METHOD checkChildAlmClass : BOOL
//------------------------------------------------------------------------------------------------------
// check child alarm classes
// set me alarm class active if at least one child has an EOFF
IF CheckAllChildAlmClass(E_AlmClass.EOFF) THEN
	CIf.Job.eMe_ActivAlmClass := E_AlmClass.EOFF;
	me.Alarm.bolfp := TRUE;
ELSIF CheckAllChildAlmClass(E_AlmClass.OFF) THEN
	CIf.Job.eMe_ActivAlmClass := E_AlmClass.OFF;
	me.Alarm.bolfp := TRUE;
ELSIF CheckAllChildAlmClass(E_AlmClass.STOP) THEN  // FB_MER needs alarm class STOP
	CIf.Job.eMe_ActivAlmClass := E_AlmClass.STOP;
	me.Alarm.bolfp := TRUE;
ELSE
	IF (me.Alarm.bolfp) THEN
		CIf.Job.eMe_ActivAlmClass := E_AlmClass.NONE; // no reset necessary
		me.Alarm.bolfp := FALSE;
	END_IF
END_IF

//------------------------------------------------------------------------------------------------------
// set alarm class parent of childs
//------------------------------------------------------------------------------------------------------
// set alarm class parent of childs in the case of a parent EOFF or me=OFF or EOFF
IF (CIf.Job.eParent_ActivAlmClass=E_AlmClass.EOFF) THEN
	SetAllChildAlmClass(CIf.Job.eParent_ActivAlmClass);
ELSIF(CIf.Job.eMe_ActivAlmClass=E_AlmClass.EOFF) OR (CIf.Job.eMe_ActivAlmClass=E_AlmClass.OFF) THEN
	SetAllChildAlmClass(CIf.Job.eMe_ActivAlmClass);
ELSE
	// no important alarm for child active
	SetAllChildAlmClass(E_AlmClass.NONE);
END_IF
END_METHOD

METHOD PROTECTED checkChildValid : BOOL
IF (usiNumOfLines = usiNumOfValidPointerToLine) THEN
	checkChildValid:= TRUE;
ELSE
	checkChildValid:= FALSE;
	// Invalid child pointer
	IF (usiNumOfLines <> usiNumOfValidPointerToLine) THEN
		// SIf.Alm[1].strText := 'Invalid child pointer'; 
		pfbAlarmCtrl^.setAlarm(CIf.Info.intCtrlId,1,0,ADR(SIf.Alm),E_AlmState.RST,CIf.Job.eMe_ActivAlmClass);	
	END_IF
END_IF
END_METHOD

METHOD PROTECTED checkStateAllLines : BOOL
VAR_INPUT
	cSTA: INT;
END_VAR
VAR
	ii: INT;
	usiNumOfCheckedChilds: USINT;
END_VAR
// Method check input state of all lines

//Init
checkStateAllLines:= FALSE;
usiNumOfCheckedChilds:= 0;

// Loop over all childs
FOR ii:=0 TO usiNumOfLines-1 BY 1 DO
	// Check state	
	// Special condition: In case if the child is in state ERROR and STOP is requested. Set child as checked.
	// Parent controller need state STOP that automatic stop sequence can work for all other childs.
	IF (a_pLineChildCIF[ii]^.Job.intState = cSTA) OR ((a_pLineChildCIF[ii]^.Job.intState = cSTA_ERROR) AND (cSTA = cSTA_STOP)) THEN
		usiNumOfCheckedChilds:= usiNumOfCheckedChilds+1;
		SIf.Cur.a_bolChildReady[ii] := TRUE;
	ELSE
		SIf.Cur.a_bolChildReady[ii] := FALSE;		
	END_IF

END_FOR

// All states equal the input state
IF (usiNumOfCheckedChilds = usiNumOfLines) THEN
	checkStateAllLines:= TRUE;
END_IF
END_METHOD

METHOD PROTECTED CmdToAllLines
VAR_INPUT
	cCMD: INT;
END_VAR
VAR
	ii: INT;
END_VAR
// Method send input command to all existing line child controller.
FOR ii:=0 TO usiNumOfLines-1 BY 1 DO	
	a_pLineChildCIF[ii]^.Job.intACmd:= cCMD;
END_FOR
END_METHOD

METHOD PROTECTED CtrlInit : BOOL
VAR
	ii: INT;
END_VAR
SUPER^.CtrlInit();

//----------------------------------------------------------------------
// Initialize all lines
//----------------------------------------------------------------------

// Method initialize all line child controller.
FOR ii:=0 TO usiNumOfLines-1 BY 1 DO	
	a_pLineChildCIF[ii] := THIS^.AddChild(a_pLineChildCtrl[ii]^);
	a_pLineChildSIF[ii] := a_pLineChildCtrl[ii]^.getCtrlSIf();
END_FOR
END_METHOD

METHOD FB_init : BOOL
VAR_INPUT
	///if TRUE, the retain variables are initialized (warm start / cold start)
	bInitRetains: BOOL;
	///if TRUE, the instance afterwards gets moved into the copy code (online change)
	bInCopyCode: BOOL;
END_VAR
VAR
	ii: UINT;
END_VAR
//------------------------------------------------------------------------------------------------------------------------
// to manually change in new FUB implementation!!!
// define valid commands for this controller
FOR ii:= 0 TO (SIZEOF(CIf.Job.aCmdList)/SIZEOF(CIf.Job.aCmdList[0])-1) BY 1 DO
	IF (CIf.Job.aCmdList[ii].intCmd=cCMD_INITIALIZED) THEN
		// found first empty array element
		EXIT;
	END_IF
END_FOR

CIf.Job.aCmdList[ii].intCmd := cCMD_STOP;
CIf.Job.aCmdList[ii].strName := 'Stop'; 
CIf.Job.aCmdList[ii].bolAvailable := TRUE;
ii := ii +1;
CIf.Job.aCmdList[ii].intCmd := cCMD_RUN;
CIf.Job.aCmdList[ii].strName := 'Run';
CIf.Job.aCmdList[ii].bolAvailable := TRUE;

// set name of class/typ
CIf.Info.strType := 'FB_MER'; 

// set alarm class
SIf.Alm[1].eAlmClass := E_AlmClass.STOP;
SIf.Alm[1].strText := 'Invalid child pointer';
SIf.Alm[2].eAlmClass := E_AlmClass.INFO;
SIf.Alm[2].strText := 'Invalid line number. Line not exist';
SIf.Alm[3].eAlmClass := E_AlmClass.INFO;
SIf.Alm[3].strText := 'Merger waits for jam sensor free'; 


//*******************************************************************************
// initial values
//*******************************************************************************

// software configuration
CIf.SwCfg.bolExist := TRUE;
CIf.SwCfg.bolSimulation := FALSE;

// configuration
SIf.Cfg.usiMergeMainMode:= E_Typ_MER_MODE.Automatic;
SIf.Cfg.usiCountJamSensors:= 0;

// parameter
SIf.Par.udi_jamTimeout_ms:= 500;
FOR ii:= 0 TO Base_PLC.cMaxNrOfChilds DO
	SIf.Par.a_bolEnableHangerRelease[ii] := TRUE;
END_FOR
// Default parameter for the lines are set in method InitLines
END_METHOD

METHOD PROTECTED getCmdState : STRING
VAR_INPUT
	intCmdState: INT;
	bolState: BOOL;
END_VAR
getCmdState := SUPER^.getCmdState(intCmdState:=intCmdState,bolState:=bolState); // get global/base defined cmds/states
IF (getCmdState='') THEN // global not defined get local
	// get string cmd/state string information in runtime
	IF (bolState=FALSE) THEN
		// cmd's
		CASE intCmdState OF
		END_CASE;
	ELSE
	
	// states
		CASE intCmdState OF	
			// SUB States
			cSTA_SUB_INITIALIZED:
				getCmdState := 'cSTA_SUB_INITIALIZED';			
			cSTA_SUB_WAIT_FOR_CMD:
				getCmdState := 'cSTA_SUB_WAIT_FOR_CMD';					
			cSTA_SUB_CHECK_HANGER_EXIST:
				getCmdState := 'cSTA_SUB_CHECK_HANGER_EXIST';
			cSTA_SUB_SEND_RELEASE:
				getCmdState := 'cSTA_SUB_SEND_RELEASE';
			cSTA_SUB_SEND_RELEASE_ALL:
				getCmdState := 'cSTA_SUB_SEND_RELEASE_ALL';	
			cSTA_SUB_SEND_STOP:
				getCmdState := 'cSTA_SUB_SEND_STOP';		
			cSTA_SUB_WAIT_JOB_DONE:
				getCmdState := 'cSTA_SUB_WAIT_JOB_DONE';
			cSTA_SUB_CHECK_MERGE_CON:
				getCmdState := 'cSTA_SUB_CHECK_MERGE_CON';
			cSTA_SUB_WAIT_LINE_FREE:
				getCmdState := 'cSTA_SUB_WAIT_LINE_FREE';	
			cSTA_SUB_END:
				getCmdState := 'cSTA_SUB_END';	
		END_CASE;
	END_IF
END_IF
END_METHOD

METHOD getCtrlSIf : POINTER TO T_Ctrl_SIf_MER
getCtrlSIf := ADR(SIf);
END_METHOD

METHOD PROTECTED IoInBridge : BOOL
// digitale and analoge inputs read from hardware or forcing
// Read sensors for waiting if a jam is detected
FOR intI := 1 TO SIf.Cfg.usiCountJamSensors DO
	SIf.In.a_bolJamSensor[intI].map := THIS^.In_a_bolJamSensor[intI];
	IF (CIf.SwCfg.bolSimulation = FALSE) THEN
		getInBol(CIf.Job.bolIoForce,ADR(SIf.In.a_bolJamSensor[intI]));
	END_IF
END_FOR

IF (CIf.SwCfg.bolSimulation = FALSE) THEN
	//ctrl.In.bol_PosSwitchBasicDefTyp.intern := getInBol(ctrl.ifc.Job.bol_Force ,ADR(ctrl.In.bol_PosSwitchBasicDefTyp);
ELSE
	//simulation of global IO
END_IF
END_METHOD

METHOD PROTECTED IoOutBridge : BOOL
// digitale and analoge inputs read from hardware or forcing

// ... no physical outputs

IF (CIf.SwCfg.bolSimulation = FALSE) THEN
	// check interlocks to prevent damages
	IF (CIf.Job.bolIlkOverwrite=FALSE) THEN
		;
	END_IF
END_IF
END_METHOD

PROPERTY MaxCapacity : DINT
GET
MaxCapacity:= SIf.Cur.dinMaxCapacity;
END_GET
END_PROPERTY

PROPERTY NumOfHangers : DINT
GET
NumOfHangers:= SIf.Cur.dinCurrentItemCount;
END_GET
END_PROPERTY

METHOD PROTECTED sta_OFF : BOOL
// state implemetation
//--------------------------------------------------------------------------------------
// Entry action
	IF (me.StateMachine.intState<>me.StateMachine.intStateLastCycle) THEN
		me.StateMachine.intStateLastCycle := me.StateMachine.intState;
		;		
	END_IF

//--------------------------------------------------------------------------------------
// Cyclic action
	IF (me.StateMachine.intState=me.StateMachine.intStateLastCycle) THEN
		
		// Reset total counter
		SIf.Cur.dinNumOfMergedHangersTotal:= 0;
		
		// State Change Condition
		IF (me.Alarm.eActivAlmClass<>E_AlmClass.EOFF) AND (me.Alarm.eActivAlmClass<>E_AlmClass.OFF) THEN
			IF (me.intCmd=cCMD_STOP) THEN
				me.StateMachine.intStateNext := cSTA_STOPBusy;
			ELSIF (me.intCmd=cCMD_RUN) THEN 
				me.StateMachine.intStateNext := cSTA_RUNBusy;
			END_IF
		END_IF
	END_IF

//--------------------------------------------------------------------------------------
// Exit action
	IF (me.StateMachine.intState<>me.StateMachine.intStateNext) THEN
		;
	END_IF
END_METHOD

METHOD PROTECTED sta_RUN : BOOL
// state implemetation
//--------------------------------------------------------------------------------------
// Entry action
	IF (me.StateMachine.intState<>me.StateMachine.intStateLastCycle) THEN
		me.StateMachine.intStateLastCycle := me.StateMachine.intState;	
		;
	END_IF

//--------------------------------------------------------------------------------------
// Cyclic action
	IF (me.StateMachine.intState=me.StateMachine.intStateLastCycle) THEN
			
	
		// Check States for parent information
		THIS^.checkStateAllLines(cSTA_RUN);

		// Check jam detection
		IF (udiJamReleaseDelayTime_ms > SIf.Par.udi_jamTimeout_ms) THEN
			bolJamDetected := FALSE;
		ELSE
			udiJamReleaseDelayTime_ms := udiJamReleaseDelayTime_ms + me.FUBInfo.udiSample_ms;
		END_IF
		
		FOR intI := 1 TO SIf.Cfg.usiCountJamSensors DO
			// Start jam timer
			IF ((SIf.In.a_bolJamSensor[intI].intern = TRUE) AND (a_bolJamSensorOnce[intI] = FALSE)) THEN
				a_bolJamSensorOnce[intI]:= TRUE;
				//a_udiTimeJamDetection[intI]:= me.StateMachine.udiTimeInState_ms;
				a_udiTimeJamDetection[intI]:= 0;
			// Stop jam timer
			ELSIF ((SIf.In.a_bolJamSensor[intI].intern = FALSE) AND (a_bolJamSensorOnce[intI] = TRUE)) THEN
				a_bolJamSensorOnce[intI]:= FALSE;
			// Set flag if neccessary
			ELSIF ((SIf.In.a_bolJamSensor[intI].intern = TRUE) AND (a_bolJamSensorOnce[intI] = TRUE)) THEN
				//IF (me.StateMachine.udiTimeInState_ms > a_udiTimeJamDetection[intI] + SIf.Par.udi_jamTimeout_ms) THEN
				IF (a_udiTimeJamDetection[intI] > SIf.Par.udi_jamTimeout_ms) THEN
					bolJamDetected := TRUE;
					udiJamReleaseDelayTime_ms := 0;
				END_IF
			END_IF
			a_udiTimeJamDetection[intI]:= a_udiTimeJamDetection[intI]+ me.FUBInfo.udiSample_ms;
		END_FOR
	
		//----------------------------------------------------------------------------------------
		// Substates for merging lines dependent time or distribution of the number of hangers
		//----------------------------------------------------------------------------------------
		CASE me.SubStateMachine.intState OF
	
			//-----------------------------------------------
			// INITIALIZE 					(MODE: All modes)
			//-----------------------------------------------
			cSTA_SUB_INITIALIZED:
			
				// Check configured main mode
				CASE SIf.Cfg.usiMergeMainMode OF	
				
					// Mode - Automatic
					E_Typ_MER_MODE.Automatic:		
						me.SubStateMachine.intStateNext := cSTA_SUB_CHECK_HANGER_EXIST;					
									
					// Mode - OnCommand	
					E_Typ_MER_MODE.OnCommand:		
						me.SubStateMachine.intStateNext := cSTA_SUB_WAIT_FOR_CMD;
														
				END_CASE
			
			//-----------------------------------------------
			// WAIT FOR COMMAND 			(MODE: OnCommand)
			//-----------------------------------------------	
			cSTA_SUB_WAIT_FOR_CMD:
			
				// Wait for command to release all
				IF (me.intCmd=SLB_CmdState.cCMD_RELEASE_ALL) THEN
					// Check about valid line number
					IF ((SIf.Par.usiLineNumToReleaseAll = 0) OR (SIf.Par.usiLineNumToReleaseAll > usiNumOfLines)) THEN
						// Invalid line	
						// SIf.Alm[2].strText := 'Invalid line number. Line not exist'; 
						pfbAlarmCtrl^.setAlarm(CIf.Info.intCtrlId,2,0,ADR(SIf.Alm),E_AlmState.RST,CIf.Job.eMe_ActivAlmClass);		
					ELSE
						// Valid line	
						usiLineNumToReleaseAll:= SIf.Par.usiLineNumToReleaseAll-1;
						me.SubStateMachine.intStateNext := cSTA_SUB_SEND_RELEASE_ALL;
					END_IF
						
				END_IF
				
			//-----------------------------------------------
			// CHECK HANGER EXIST 			(MODE: Automatic)     
			//-----------------------------------------------
			cSTA_SUB_CHECK_HANGER_EXIST:
				// Entry action
				IF (me.SubStateMachine.intState<>me.SubStateMachine.intStateLastCycle) THEN
					me.SubStateMachine.intStateLastCycle := me.SubStateMachine.intState;							
					;						
				END_IF
				
				// Init
				bolReleaseHanger:= FALSE;
					
				// Check hanger exists on line
				IF (a_pLineChildSIF[usiIndexToRelease]^.Cur.bolHangerDetected=TRUE) AND 
					(Sif.par.a_bolEnableHangerRelease[usiIndexToRelease] = TRUE) THEN		// MRU added
					bolReleaseHanger:= TRUE;					
				ELSE		
					// No hanger on this line, check next
					IF (usiIndexToRelease < (usiNumOfLines-1)) THEN
						// Inc. index to next line
						usiIndexToRelease:= usiIndexToRelease + 1;	
					ELSE
						usiIndexToRelease:= 0;
					END_IF
				END_IF			
	
				// State Change Condition
				IF (bolReleaseHanger=TRUE) THEN
					me.SubStateMachine.intStateNext := cSTA_SUB_SEND_RELEASE;
					// Reset counter and timer
					dinNumOfPassedHangers:=0;
					udiMergingTime:=0;
				END_IF
					
			//-----------------------------------------------
			// SEND RELEASE					(MODE: Automatic)
			//-----------------------------------------------
			cSTA_SUB_SEND_RELEASE:		
	
				// Send release command to line X (trigger command)
				a_pLineChildCIF[usiIndexToRelease]^.Job.intACmd:= STB_CmdState.cCMD_RELEASE;				
				
				// State Change Condition
				IF(TRUE)THEN
					me.SubStateMachine.intStateNext := cSTA_SUB_WAIT_JOB_DONE;					
				END_IF	
						
			//-----------------------------------------------
			// SEND RELEASE	ALL				(MODE: OnCommand)
			//-----------------------------------------------
			cSTA_SUB_SEND_RELEASE_ALL:
			
				// Send release all command to line X
				a_pLineChildCIF[usiLineNumToReleaseAll]^.Job.intACmd:= STB_CmdState.cCMD_RELEASE_ALL;				
				
				// State Change Condition
				IF(TRUE)THEN
					me.SubStateMachine.intStateNext := cSTA_SUB_WAIT_JOB_DONE;					
				END_IF		
					
			//-----------------------------------------------
			// WAIT JOB DONE				(MODE: All modes)
			//-----------------------------------------------
			cSTA_SUB_WAIT_JOB_DONE:
		
				// Check configured main mode
				CASE SIf.Cfg.usiMergeMainMode OF	
				
					// Mode - Automatic
					E_Typ_MER_MODE.Automatic:
						// State Change Condition
						// Wait until job done
						IF(a_pLineChildCIF[usiIndexToRelease]^.Job.intACmd = cSTA_DONE) THEN									
							me.SubStateMachine.intStateNext := cSTA_SUB_CHECK_MERGE_CON;																				
						END_IF	
									
					// Mode - OnCommand	
					E_Typ_MER_MODE.OnCommand:
						// State Change Condition
						// Wait until release all
						IF(a_pLineChildCIF[usiLineNumToReleaseAll]^.Job.intState = SLB_CmdState.cCMD_RELEASE_ALL)THEN				
							me.SubStateMachine.intStateNext := cSTA_SUB_SEND_STOP;																
						END_IF
						
				END_CASE
							
			//-----------------------------------------------
			// SEND STOP					(MODE: OnCommand)
			//-----------------------------------------------
			cSTA_SUB_SEND_STOP:
			
				// Send stop command to line X
				a_pLineChildCIF[usiLineNumToReleaseAll]^.Job.intACmd:=cCMD_RUN;				
				
				// State Change Condition
				IF(a_pLineChildCIF[usiLineNumToReleaseAll]^.Job.intState=cSTA_RUN)THEN
					me.SubStateMachine.intStateNext := cSTA_SUB_WAIT_LINE_FREE;					
				END_IF	
								
			//-----------------------------------------------
			// CHECK MERGE CONDITIONS		(MODE: Automatic)
			//-----------------------------------------------
			cSTA_SUB_CHECK_MERGE_CON:
				// Entry action
				IF (me.SubStateMachine.intState<>me.SubStateMachine.intStateLastCycle) THEN
					me.SubStateMachine.intStateLastCycle := me.SubStateMachine.intState;							
					;						
				END_IF
					
				// Count the passed hangers from current line X
				IF (a_pLineChildSIF[usiIndexToRelease]^.Cur.dinHangersPassedTotal <> dinPassedTotalLineXOld) THEN
					// Count passed hangers if "E_Typ_MER_AUTO_MODE.MergeOverSetpoint" is selected.				
					dinNumOfPassedHangers:= dinNumOfPassedHangers + a_pLineChildSIF[usiIndexToRelease]^.Cur.uinNumOfHangersPerPulseFirstZone;			
					// Calculate merged hangers total
					SIf.Cur.dinNumOfMergedHangersTotal:= SIf.Cur.dinNumOfMergedHangersTotal + a_pLineChildSIF[usiIndexToRelease]^.Cur.uinNumOfHangersPerPulseFirstZone;									
				END_IF
				dinPassedTotalLineXOld:= a_pLineChildSIF[usiIndexToRelease]^.Cur.dinHangersPassedTotal;
		
					
				// State Change Condition
				IF (a_pLineChildSIF[usiIndexToRelease]^.Cur.bolHangerDetected=FALSE) THEN	// No hanger exist
					me.SubStateMachine.intStateNext := cSTA_SUB_WAIT_LINE_FREE;				
				ELSIF ((SIf.Par.a_LinePar[usiIndexToRelease].usiMergeMode = E_Typ_MER_AUTO_MODE.MergeOverTime) AND (udiMergingTime >= SIf.Par.a_LinePar[usiIndexToRelease].udiMergingTime_ms)) THEN
					me.SubStateMachine.intStateNext := cSTA_SUB_WAIT_LINE_FREE;				
				ELSIF ((SIf.Par.a_LinePar[usiIndexToRelease].usiMergeMode = E_Typ_MER_AUTO_MODE.MergeOverSetpoint) AND (dinNumOfPassedHangers >= SIf.Par.a_LinePar[usiIndexToRelease].uinNumOfHangersToMerge)) THEN
					me.SubStateMachine.intStateNext := cSTA_SUB_WAIT_LINE_FREE;							
				ELSIF ((SIf.Par.a_LinePar[usiIndexToRelease].usiMergeMode = E_Typ_MER_AUTO_MODE.MergeOverTime) AND (udiMergingTime < SIf.Par.a_LinePar[usiIndexToRelease].udiMergingTime_ms)) THEN
					me.SubStateMachine.intStateNext := cSTA_SUB_SEND_RELEASE;					
				ELSIF ((SIf.Par.a_LinePar[usiIndexToRelease].usiMergeMode = E_Typ_MER_AUTO_MODE.MergeOverSetpoint) AND (dinNumOfPassedHangers < SIf.Par.a_LinePar[usiIndexToRelease].uinNumOfHangersToMerge)) THEN
					me.SubStateMachine.intStateNext := cSTA_SUB_SEND_RELEASE;	
				END_IF
	
			//-----------------------------------------------
			// WAIT UNTIL LINE IS FREE		(MODE: All modes)
			//-----------------------------------------------
			cSTA_SUB_WAIT_LINE_FREE:

				IF (bolJamDetected	= TRUE) THEN // Line is not free, jam detected
					// SIf.Alm[3].strText := 'Merger waits for jam sensor free';
					pfbAlarmCtrl^.setAlarm(CIf.Info.intCtrlId,3,0,ADR(SIf.Alm),E_AlmState.RST,CIf.Job.eMe_ActivAlmClass);				
				ELSE				
					// Check configured main mode
					CASE SIf.Cfg.usiMergeMainMode OF	
					
						// Mode - Automatic
						E_Typ_MER_MODE.Automatic:
							// State Change Condition
							IF (me.SubStateMachine.udiTimeInState_ms > SIf.Par.a_LinePar[usiIndexToRelease].udiWaitTimeLineFree_ms) THEN 
								IF(me.intCmd=cCMD_STOP)THEN
									// Go to end
									me.SubStateMachine.intStateNext := cSTA_SUB_END;
								ELSE
									// Merging cycle line X complete
									IF (usiIndexToRelease < (usiNumOfLines-1)) THEN						
										// Inc. index to next line
										usiIndexToRelease:= usiIndexToRelease + 1;	
									ELSE
										usiIndexToRelease:= 0;
									END_IF
									
									// Go on with automatic cycle
									me.SubStateMachine.intStateNext := cSTA_SUB_CHECK_HANGER_EXIST;					
								END_IF		
							END_IF
									
						// Mode - OnCommand	
						E_Typ_MER_MODE.OnCommand:
							// State Change Condition
							IF (me.SubStateMachine.udiTimeInState_ms > SIf.Par.a_LinePar[usiLineNumToReleaseAll].udiWaitTimeLineFree_ms) THEN												
								// Update merged hangers total -> After release all, use passed package 
								SIf.Cur.dinNumOfMergedHangersTotal:= SIf.Cur.dinNumOfMergedHangersTotal + a_pLineChildSIF[usiLineNumToReleaseAll]^.Cur.dinHangersPassedPackage;			
								
								IF(me.intCmd=cCMD_STOP)THEN
									// Go to end
									me.SubStateMachine.intStateNext := cSTA_SUB_END;
								ELSE
									//Set "Job done" for parent
									CIf.Job.intACmd:=cSTA_DONE;
									me.SubStateMachine.intStateNext := cSTA_SUB_WAIT_FOR_CMD;
								END_IF								
							END_IF
							
					END_CASE
				END_IF
			//-----------------------------------------------
			// END							(MODE: All modes)
			//-----------------------------------------------
			cSTA_SUB_END:
			     // ... do nothing
		
		END_CASE

		// Timer handling for merging time
		udiMergingTime:= udiMergingTime + me.FUBInfo.udiSample_ms;
			
		// State Change Condition
		IF ((me.intCmd=cCMD_STOP) AND ((me.SubStateMachine.intState=cSTA_SUB_END) OR (me.SubStateMachine.intState=cSTA_SUB_CHECK_HANGER_EXIST) OR (me.SubStateMachine.intState=cSTA_SUB_WAIT_FOR_CMD) OR (me.SubStateMachine.intState=cSTA_SUB_WAIT_LINE_FREE))) THEN
			me.StateMachine.intStateNext := cSTA_STOPBusy;
		END_IF
	END_IF

//--------------------------------------------------------------------------------------
// Exit action
	IF (me.StateMachine.intState<>me.StateMachine.intStateNext) THEN
		;
	END_IF
END_METHOD

METHOD PROTECTED sta_RUNBusy : BOOL
VAR
	ii: INT;
END_VAR
// state implemetation
//--------------------------------------------------------------------------------------
// Entry action
	IF (me.StateMachine.intState<>me.StateMachine.intStateLastCycle) THEN
		me.StateMachine.intStateLastCycle := me.StateMachine.intState;
	
		bolGoToRun:= FALSE;
		usiIndexToRelease:= 0;
		
		// Initialize sub state machine
		me.SubStateMachine.intState:= cSTA_SUB_INITIALIZED; 
		me.SubStateMachine.intStateNext:= cSTA_SUB_INITIALIZED;
		
	END_IF

//--------------------------------------------------------------------------------------
// Cyclic action
	IF (me.StateMachine.intState=me.StateMachine.intStateLastCycle) THEN
					
		// Check configured main mode
		CASE SIf.Cfg.usiMergeMainMode OF	
		
			// Mode - Automatic
			E_Typ_MER_MODE.Automatic:
			
				// send command RUN to all existing line child controller.
				THIS^.CmdToAllLines(cCMD_RUN);
				
				// State Change Condition
				// Check if all childs in "RUN", ready for release hanger 
				IF(THIS^.checkStateAllLines(cSTA_RUN))THEN
					bolGoToRun:= TRUE;			
				END_IF	
		
			// Mode - OnCommand	
			E_Typ_MER_MODE.OnCommand:
			
				// send command STOP to all existing line child controller.
				THIS^.CmdToAllLines(cCMD_RUN);
				
				// State Change Condition
				// Check if all childs stopped, ready for new command 
				IF(THIS^.checkStateAllLines(cSTA_RUN))THEN
					bolGoToRun:= TRUE;					
				END_IF	
			
		END_CASE

	
		// State Change Condition	
		IF (bolGoToRun=TRUE) THEN
			me.StateMachine.intStateNext := cSTA_RUN;		
		END_IF

	END_IF

//--------------------------------------------------------------------------------------
// Exit action
	IF (me.StateMachine.intState<>me.StateMachine.intStateNext) THEN
		;
	END_IF
END_METHOD

METHOD PROTECTED sta_STOP : BOOL
// state implemetation
//--------------------------------------------------------------------------------------
// Entry action
	IF (me.StateMachine.intState<>me.StateMachine.intStateLastCycle) THEN
		me.StateMachine.intStateLastCycle := me.StateMachine.intState;
		;
	END_IF

//--------------------------------------------------------------------------------------
// Cyclic action
	IF (me.StateMachine.intState=me.StateMachine.intStateLastCycle) THEN

		// State Change Condition	
		IF (me.intCmd = cCMD_RUN) THEN 
			me.StateMachine.intStateNext := cSTA_RUNBusy;
		END_IF
	END_IF

//-------------------------------------------------------------------------------------
// Exit action
	IF (me.StateMachine.intState<>me.StateMachine.intStateNext) THEN
		;
	END_IF
END_METHOD

METHOD PROTECTED sta_STOPBusy : BOOL
// state implemetation
//--------------------------------------------------------------------------------------
// Entry action
	IF (me.StateMachine.intState<>me.StateMachine.intStateLastCycle) THEN
		me.StateMachine.intStateLastCycle := me.StateMachine.intState;
		
		// send command STOP to all existing line child controller.
		THIS^.CmdToAllLines(cCMD_STOP);

	END_IF

//--------------------------------------------------------------------------------------
// Cyclic action
	IF (me.StateMachine.intState=me.StateMachine.intStateLastCycle) THEN
			
		// State Change Condition
		// Check if all STOPPED
		IF (THIS^.checkStateAllLines(cSTA_STOP)) THEN
			me.StateMachine.intStateNext := cSTA_STOP;
		END_IF
	END_IF

//--------------------------------------------------------------------------------------
// Exit action
	IF (me.StateMachine.intState<>me.StateMachine.intStateNext) THEN
		;
	END_IF
END_METHOD

METHOD PROTECTED StateMachine : BOOL
SUPER^.StateMachine();

// main statemachine of base controller
CASE me.StateMachine.intState OF
    cSTA_STOPBusy: 
        THIS^.sta_STOPBusy();
    cSTA_STOP: 
        THIS^.sta_STOP();
	cSTA_RUNBusy: 
        THIS^.sta_RUNBusy();
    cSTA_RUN: 
        THIS^.sta_RUN();				
END_CASE;
END_METHOD

END_FUNCTION_BLOCK

// POUs/Controller/Lvl1/SLB (Slide buffer)/FB_SLB
FUNCTION_BLOCK FB_SLB EXTENDS FB_CtrlBase IMPLEMENTS IBuffer
VAR
	/// Specific interface struct for public access
	SIf: T_Ctrl_SIf_SLB;
	/// List of pointers to Childs
	a_pBufferZoneChildCtrl: ARRAY[0..Base_Const.cMaxNrOfChilds] OF POINTER TO FB_STB;
	/// List of childs common interface
	a_pBufferZoneChildCIF: ARRAY[0..Base_Const.cMaxNrOfChilds] OF POINTER TO T_Ctrl_CIf;
	/// List of childs specific interface for additional parameters or cur
	a_pBufferZoneChildSIF: ARRAY[0..Base_Const.cMaxNrOfChilds] OF POINTER TO T_Ctrl_SIf_STB;
	/// Function specific variables
	usiNumOfBufferZones: USINT;
	usiNumOfValidPointerToZone: USINT;
	bolAllZonesEmpty: BOOL;
	dinPassedTotalZone1Old: DINT;
	/// Var. used for sub sequence refill
	intIndexRefill: INT;
	SubStateMachineRefill: INT;
	udiTimeInStateRefill_ms: UDINT;
	// Array used in RefillZones_parallel
	a_udiTimeInStateRefill_ms: ARRAY [0..Base_Const.cMaxNrOfChilds] OF UDINT;
	/// Var. used for simulation
	abolRESimRetract: ARRAY[0..Base_Const.cMaxNrOfChilds] OF BOOL;
END_VAR
VAR CONSTANT
	/// sub States
	cSTA_SUB_WAIT_FOR_CMD: INT := 500;
	cSTA_SUB_SEND_RELEASE: INT := 502;
	cSTA_SUB_SEND_STOP: INT := 504;
	cSTA_SUB_BREAK: INT := 506;
END_VAR

(*__________________________________________________________________________________________________
¦	
¦	Vistaprint Schweiz GmbH
¦	CH - 8401 Winterthur
¦
¦	www.vistaprint.ch - info@vistaprint.ch
¦___________________________________________________________________________________________________

Function desription:
The slide buffer controller handles the automatic refill and sequential emptying of different buffer zones. 
Buffer zones may consist of the following components: Separator, Double Stopper or Single Stopper.

History:
Version		Date			Author		Comment
---------------------------------------------------------------------------------------------------
0.00.1		02.09.2013		AVME/DSC	Start history. 
0.00.2		04.09.2013		AVME/DSC	Integration of all slide buffer basic functionalities. 
										Test on simulator.
0.00.3		06.09.2013		AVME/DSC    Renaming of method checkChildPointer to checkChildValid.
										Insert add. validation to check if the number of added childs is valid.
										Slide buffer controller can now also used with only one buffer.
0.00.4 		09.09.2013		AVME/DSC    Copied content from state "RUN_busy" to "RUN".  
										Insert new method for calculation of the max. capacity for all childs.
0.00.5		10.09.2013		AVME/PRE	Implement Simulation
										Correct counter if buffer empty only if hanger detection sensor
										Give released item to next Buffer
0.00.6		19.09.2013		AVME/PRE	Implement new Base Concept
0.00.7		28.10.2013		VP/RE		SLB is full is last zone is full. Otherwise it leads to overflow problems.
0.00.8 		04.11.2013		AVME/DSC    Modified ".cur" interface. Newly distinction is made ​​between: "bolInputBufferFull" and  "bolAllBuffersFull"
0.00.9		03.12.2013		AVME/MRU	Add MaxCapacity / NumOfHangers properties
0.00.10		09.12.2013		AVME/DSC	Modification in method "checkStateAllZones".
										Special condition: In case if the child is in state ERROR and STOP is requested. Set child as checked.
										Parent controller need state STOP that automatic stop sequence can work for all other childs.
0.00.11		10.01.2014		AVME/MRU	Bugzilla ID 55: Refill aloud, if dinNumOfHangersInBuffer < dinMaxCapacity (Without uinNumOfHangersPerPulse)
0.00.12		13.01.2014		AVME/MRU	Bugzilla ID 03: BufferFull for LineControl added
0.00.13		30.06.2014		AVME/MRU	RefillZones_parallel added
										
__________________________________________________________________________________________________*)


IF ((me.bolActivate) AND (THIS^.checkChildValid())) THEN // cyclic call enabled
	IF (CIf.Info.bolInitDone=FALSE) THEN // first cycle -> init
		CtrlInit();
		CIf.Info.bolInitDone := TRUE;
	ELSE
		CycleStartDuty();
	
		Always();
		
		StateMachine();
		
		CycleEndDuty();
	END_IF
END_IF;

METHOD AddBufferZone
VAR_INPUT
	p_BufferZone: POINTER TO FB_STB;
END_VAR

// Method add the pointer address of the buffer zone child controller to the array list.
IF (usiNumOfBufferZones <= (Base_Const.cMaxNrOfChilds-1)) THEN
	// Add buffer zone child controller to list
	a_pBufferZoneChildCtrl[usiNumOfBufferZones] := p_BufferZone;
	// Inc. number of buffer zones
	usiNumOfBufferZones:= usiNumOfBufferZones+1;
	// Check if the pointer is valid
	IF (p_BufferZone<>0) THEN
		usiNumOfValidPointerToZone:= usiNumOfValidPointerToZone+1;
	END_IF
END_IF
END_METHOD

METHOD PROTECTED Always : BOOL
IF (me.bolChangeBackToAUTO=TRUE) THEN // switch mode to automatic switch off controller
	//me.StateMachine.intStateNext := cSTA_OFFBusy;
	//me.bolChangeBackToAUTO := FALSE; // for cylinder no change to off when switch to automatic!!
END_IF

SUPER^.Always();

// ----------------------------------------------------------------------------------
// cyclic actions outside of statemachine
IF (me.StateMachine.intState<>cSTA_SINGLE_ANSWER) THEN
	
	//-------------------------------------------------
	// Provide current values for the parent
	//-------------------------------------------------	
	
	// Number of buffer zones, depends on how many times the method "AddBufferZone" was called at init
	SIf.Cur.usiNumOfBufferZones:= usiNumOfBufferZones;
	// Input buffer is full -> based on last zone full signal
	SIf.Cur.bolInputBufferFull := a_pBufferZoneChildSIF[usiNumOfBufferZones-1]^.Cur.bolBufferFull;	
	// All buffers full -> based on all zones
	SIf.Cur.bolAllBuffersFull:= THIS^.checkAllZonesFull();
	// Approximate number of hangers in buffer -> based on all zones
	SIf.Cur.dinNumOfHangersInBuffer:= THIS^.CalcSumNumOfHangers();
	// Max. buffer capacity -> based on all zones
	SIf.Cur.dinMaxCapacity:= THIS^.CalcMaxCapacity();	
	// Hangers passed total counter, always from zone 1, output
	SIf.Cur.dinHangersPassedTotal:= a_pBufferZoneChildSIF[0]^.Cur.dinHangersPassedTotal;
	// Hanger detected, always from zone 1, output
	SIf.Cur.bolHangerDetected:= a_pBufferZoneChildSIF[0]^.Cur.bolHangerDetected;
	// Number of passing hangers per pulse in first zone
	SIf.Cur.uinNumOfHangersPerPulseFirstZone:= a_pBufferZoneChildSIF[0]^.Cfg.uinNumOfHangersPerPulse;
	
	
	// Set alarm all buffer zones full
	IF (SIf.Cur.bolAllBuffersFull = TRUE) THEN	
		// SIf.Alm[3].strText := 'All buffer zones full';	 
		pfbAlarmCtrl^.setAlarm(CIf.Info.intCtrlId,3,0,ADR(SIf.Alm),E_AlmState.RST,CIf.Job.eMe_ActivAlmClass);	
	END_IF
			
END_IF

// ----------------------------------------------------------------------------------
// Conditions Always
// overrule error always from base -> no EOFF State!! in EOFF go to OFF
IF (me.StateMachine.intStateNext = cSTA_EOFFBusy) THEN
	IF (me.StateMachine.intState=cSTA_OFF) THEN
		me.StateMachine.intStateNext := cSTA_OFF;
	ELSE // stay in OFF
		me.StateMachine.intStateNext := cSTA_OFFBusy;
	END_IF
END_IF
END_METHOD

PROPERTY BufferFull : BOOL
GET
BufferFull:= SIf.Cur.bolAllBuffersFull;
END_GET
END_PROPERTY

METHOD PROTECTED CalcMaxCapacity : DINT
VAR
	ii: INT;
	dinSumMaxCapacity: DINT;
END_VAR
// Method calculate the sum of max. capacities in all zones and return the result.

//Init
CalcMaxCapacity:= 0;
dinSumMaxCapacity:= 0;

// Loop over all childs
FOR ii:=0 TO usiNumOfBufferZones-1 BY 1 DO
	// Build sum of all zones		
	dinSumMaxCapacity:= dinSumMaxCapacity + a_pBufferZoneChildSIF[ii]^.Cfg.dinMaxCapacity; 	
END_FOR

// Return result
CalcMaxCapacity:= dinSumMaxCapacity;
END_METHOD

METHOD PROTECTED CalcSumNumOfHangers : DINT
VAR
	ii: INT;
	dinSumNumOfHangers: DINT;
END_VAR
// Method calculate the sum of hangers in all zones and return the result.

//Init
CalcSumNumOfHangers:= 0;
dinSumNumOfHangers:= 0;

// Loop over all childs
FOR ii:=0 TO usiNumOfBufferZones-1 BY 1 DO
	// Build sum of all zones		
	dinSumNumOfHangers:= dinSumNumOfHangers + a_pBufferZoneChildSIF[ii]^.Cur.dinNumOfHangersInBuffer; 	
END_FOR

// Return result
CalcSumNumOfHangers:= dinSumNumOfHangers;
END_METHOD

METHOD PROTECTED checkAllZonesEmpty : BOOL
VAR
	ii: INT;
	usiNumOfEmptyZones: USINT;
END_VAR
// Method check if all zones are empty. If yes, return TRUE

//Init
checkAllZonesEmpty:= FALSE;
usiNumOfEmptyZones:= 0;

// Loop over all childs
FOR ii:=0 TO usiNumOfBufferZones-1 BY 1 DO
	// Check number of hangers in buffer zone X <= 0	
	IF (a_pBufferZoneChildSIF[ii]^.Cur.dinNumOfHangersInBuffer <= 0) THEN
		usiNumOfEmptyZones:= usiNumOfEmptyZones+1;		
	END_IF
END_FOR

// All zones empty
IF (usiNumOfEmptyZones = usiNumOfBufferZones) THEN
	checkAllZonesEmpty:= TRUE;
END_IF
END_METHOD

METHOD PROTECTED checkAllZonesFull : BOOL
VAR
	ii: INT;
	usiNumOfFullZones: USINT;
END_VAR
// Method check if all zones are full. If yes, return TRUE

//Init
checkAllZonesFull:= FALSE;
usiNumOfFullZones:= 0;

// Loop over all childs
FOR ii:=0 TO usiNumOfBufferZones-1 BY 1 DO
	// Check buffer full info of zone X	
	IF (a_pBufferZoneChildSIF[ii]^.Cur.bolBufferFull=TRUE) THEN
		usiNumOfFullZones:= usiNumOfFullZones+1;		
	END_IF
END_FOR

// All zones full
IF (usiNumOfFullZones = usiNumOfBufferZones) THEN
	checkAllZonesFull:= TRUE;
END_IF
END_METHOD

METHOD checkChildAlmClass : BOOL
//------------------------------------------------------------------------------------------------------
// check child alarm classes
// set me alarm class active if at least one child has an EOFF
IF CheckAllChildAlmClass(E_AlmClass.EOFF) THEN
	CIf.Job.eMe_ActivAlmClass := E_AlmClass.EOFF;
	me.Alarm.bolfp := TRUE;
ELSIF CheckAllChildAlmClass(E_AlmClass.OFF) THEN
	CIf.Job.eMe_ActivAlmClass := E_AlmClass.OFF;
	me.Alarm.bolfp := TRUE;
ELSIF CheckAllChildAlmClass(E_AlmClass.STOP) THEN // FB_SLB needs alarm class STOP
	CIf.Job.eMe_ActivAlmClass := E_AlmClass.STOP;
	me.Alarm.bolfp := TRUE;
ELSE
	IF (me.Alarm.bolfp) THEN
		CIf.Job.eMe_ActivAlmClass := E_AlmClass.NONE; // no reset necessary
		me.Alarm.bolfp := FALSE;
	END_IF
END_IF

//------------------------------------------------------------------------------------------------------
// set alarm class parent of childs
//------------------------------------------------------------------------------------------------------
// set alarm class parent of childs in the case of a parent EOFF or me=OFF or EOFF
IF (CIf.Job.eParent_ActivAlmClass=E_AlmClass.EOFF) THEN
	SetAllChildAlmClass(CIf.Job.eParent_ActivAlmClass);
ELSIF(CIf.Job.eMe_ActivAlmClass=E_AlmClass.EOFF) OR (CIf.Job.eMe_ActivAlmClass=E_AlmClass.OFF) THEN
	SetAllChildAlmClass(CIf.Job.eMe_ActivAlmClass);
ELSE
	// no important alarm for child active
	SetAllChildAlmClass(E_AlmClass.NONE);
END_IF
END_METHOD

METHOD PROTECTED checkChildValid : BOOL
IF ((usiNumOfBufferZones = usiNumOfValidPointerToZone) AND (usiNumOfBufferZones>=Const_SLB.cusiMinAddedChilds)) THEN
	checkChildValid:= TRUE;
ELSE
	checkChildValid:= FALSE;
	
	// Invalid child pointer
	IF (usiNumOfBufferZones <> usiNumOfValidPointerToZone) THEN
		// SIf.Alm[1].strText := 'Invalid child pointer'; 
		pfbAlarmCtrl^.setAlarm(CIf.Info.intCtrlId,1,0,ADR(SIf.Alm),E_AlmState.RST,CIf.Job.eMe_ActivAlmClass);	
	END_IF
	
 	// Invalid configuration
	IF (usiNumOfBufferZones<Const_SLB.cusiMinAddedChilds) THEN
		// SIf.Alm[2].strText := 'Invalid configuration. Slide buffer needs min. 1 buffer zone'; 
		pfbAlarmCtrl^.setAlarm(CIf.Info.intCtrlId,2,0,ADR(SIf.Alm),E_AlmState.RST,CIf.Job.eMe_ActivAlmClass);	
	END_IF
	
END_IF
END_METHOD

METHOD PROTECTED checkStateAllZones : BOOL
VAR_INPUT
	cSTA: INT;
END_VAR
VAR
	ii: INT;
	usiNumOfCheckedChilds: USINT;
END_VAR
// Method check input state of all zones

//Init
checkStateAllZones:= FALSE;
usiNumOfCheckedChilds:= 0;

// Loop over all childs
FOR ii:=0 TO usiNumOfBufferZones-1 BY 1 DO
	// Check state	
	// Special condition: In case if the child is in state ERROR and STOP is requested. Set child as checked.
	// Parent controller need state STOP that automatic stop sequence can work for all other childs.
	IF (a_pBufferZoneChildCIF[ii]^.Job.intState = cSTA) OR ((a_pBufferZoneChildCIF[ii]^.Job.intState = cSTA_ERROR) AND (cSTA = cSTA_STOP)) THEN
		usiNumOfCheckedChilds:= usiNumOfCheckedChilds+1;
	END_IF
END_FOR

// All states equal the input state
IF (usiNumOfCheckedChilds = usiNumOfBufferZones) THEN
	checkStateAllZones:= TRUE;
END_IF
END_METHOD

METHOD PROTECTED CmdToAllZones
VAR_INPUT
	cCMD: INT;
END_VAR
VAR
	ii: INT;
END_VAR
// Method send input command to all existing buffer zone child controller.
FOR ii:=0 TO usiNumOfBufferZones-1 BY 1 DO	
	a_pBufferZoneChildCIF[ii]^.Job.intACmd:= cCMD;
END_FOR
END_METHOD

METHOD PROTECTED CtrlInit : BOOL
VAR
	ii: INT;
END_VAR
SUPER^.CtrlInit();

// Initialize all lines
// Method initialize all line child controller.
FOR ii:=0 TO usiNumOfBufferZones-1 BY 1 DO	
	a_pBufferZoneChildCIF[ii] := THIS^.AddChild(a_pBufferZoneChildCtrl[ii]^);
	a_pBufferZoneChildSIF[ii] := a_pBufferZoneChildCtrl[ii]^.getCtrlSIf();
END_FOR
END_METHOD

METHOD FB_init : BOOL
VAR_INPUT
	///if TRUE, the retain variables are initialized (warm start / cold start)
	bInitRetains: BOOL;
	///if TRUE, the instance afterwards gets moved into the copy code (online change)
	bInCopyCode: BOOL;
END_VAR
VAR
	ii: UINT;
END_VAR
//------------------------------------------------------------------------------------------------------------------------
// to manually change in new FUB implementation!!!
// define valid commands for this controller
FOR ii:= 0 TO (SIZEOF(CIf.Job.aCmdList)/SIZEOF(CIf.Job.aCmdList[0])-1) BY 1 DO
	IF (CIf.Job.aCmdList[ii].intCmd=cCMD_INITIALIZED) THEN
		// found first empty array element
		EXIT;
	END_IF
END_FOR

CIf.Job.aCmdList[ii].intCmd := cCMD_STOP;
CIf.Job.aCmdList[ii].strName := 'Stop'; 
CIf.Job.aCmdList[ii].bolAvailable := TRUE;
ii := ii +1;
CIf.Job.aCmdList[ii].intCmd := cCMD_RUN;
CIf.Job.aCmdList[ii].strName := 'Run';
CIf.Job.aCmdList[ii].bolAvailable := TRUE;
ii := ii +1;
CIf.Job.aCmdList[ii].intCmd := SLB_CmdState.cCMD_RELEASE_ALL;
CIf.Job.aCmdList[ii].strName := 'Release All';
CIf.Job.aCmdList[ii].bolAvailable := TRUE;
ii := ii +1;
CIf.Job.aCmdList[ii].intCmd := STB_CmdState.cCMD_RELEASE;  //Used as trigger command in state RUN_Busy
CIf.Job.aCmdList[ii].strName := 'Release';
CIf.Job.aCmdList[ii].bolAvailable := TRUE;


// set name of class/typ
CIf.Info.strType := 'FB_SLB'; 

// set alarm class
SIf.Alm[1].eAlmClass := E_AlmClass.STOP;
SIf.Alm[1].strText := 'Invalid child pointer';
SIf.Alm[2].eAlmClass := E_AlmClass.STOP;
SIf.Alm[2].strText := 'Invalid configuration. Slide buffer needs min. 1 buffer zone'; 
SIf.Alm[3].eAlmClass := E_AlmClass.INFO;
SIf.Alm[3].strText := 'All buffer zones full';

//*******************************************************************************
// initial values
//*******************************************************************************

// software configuration
CIf.SwCfg.bolExist := TRUE;
CIf.SwCfg.bolSimulation := FALSE;

// cinfiguration
SIf.Cfg.bolRefill_parallel:= FALSE;

// parameter
SIf.Par.udiIntervalBufferEmptying_ms:= 200;
SIf.Par.udiIntervalBufferFilling_ms:= 2000;
SIf.Par.udiSimIncomingTime_ms := 20000;
END_METHOD

METHOD PROTECTED getCmdState : STRING
VAR_INPUT
	intCmdState: INT;
	bolState: BOOL;
END_VAR
getCmdState := SUPER^.getCmdState(intCmdState:=intCmdState,bolState:=bolState); // get global/base defined cmds/states
IF (getCmdState='') THEN // global not defined get local
	// get string cmd/state string information in runtime
	IF (bolState=FALSE) THEN
		// cmd's
		CASE intCmdState OF
			SLB_CmdState.cCMD_RELEASE_ALL: 
				getCmdState := 'cCMD_RELEASE_ALL';
		END_CASE;
	ELSE
	
	// states
		CASE intCmdState OF
			SLB_CmdState.cSTA_RELEASE_ALLBusy: 
				getCmdState := 'cSTA_RELEASE_ALLBusy';
			SLB_CmdState.cSTA_RELEASE_ALL: 
				getCmdState := 'cSTA_RELEASE_ALL';
		
			// SUB States
			cSTA_SUB_WAIT_FOR_CMD:
				getCmdState := 'cSTA_SUB_WAIT_FOR_CMD';
			cSTA_SUB_SEND_RELEASE:
				getCmdState := 'cSTA_SUB_SEND_RELEASE';
			cSTA_SUB_SEND_STOP:
				getCmdState := 'cSTA_SUB_SEND_STOP';
			cSTA_SUB_BREAK:
				getCmdState := 'cSTA_SUB_BREAK';
						
		END_CASE;
	END_IF
END_IF
END_METHOD

METHOD getCtrlSIf : POINTER TO T_Ctrl_SIf_SLB
getCtrlSIf := ADR(SIf);
END_METHOD

METHOD PROTECTED IoInBridge : BOOL
// digitale and analoge inputs read from hardware or forcing

// ... no physical inputs

IF (CIf.SwCfg.bolSimulation = FALSE) THEN
	;
ELSE
	//simulation of global IO
END_IF
END_METHOD

METHOD PROTECTED IoOutBridge : BOOL
// digitale and analoge inputs read from hardware or forcing

// ... no physical outputs

IF (CIf.SwCfg.bolSimulation = FALSE) THEN
	// check interlocks to prevent damages
	IF (CIf.Job.bolIlkOverwrite=FALSE) THEN
		;
	END_IF
END_IF
END_METHOD

PROPERTY MaxCapacity : DINT
GET
MaxCapacity:= SIf.Cur.dinMaxCapacity;
END_GET
END_PROPERTY

PROPERTY NumOfHangers : DINT
GET
NumOfHangers:= SIf.Cur.dinNumOfHangersInBuffer;
END_GET
END_PROPERTY

METHOD RefillZones
VAR
	/// Loop variable
	ii: INT;
END_VAR
// Simulation
fbSimulationTimer.PT := UDINT_TO_TIME(SIf.Par.udiSimIncomingTime_ms);
IF (CIf.SwCfg.bolSimulation) THEN
	// Cyclicle input into the top stopperbuffer
	fbSimulationTimer(); // set time/reset timer
	IF fbSimulationTimer.Q = TRUE THEN
		fbSimulationTimer.IN := FALSE;
		a_pBufferZoneChildSIF[usiNumOfBufferZones-1]^.In.bolBufferFull.intern := TRUE;
		IF a_pBufferZoneChildSIF[usiNumOfBufferZones-1]^.Cfg.bolHasBufferFullSensor = FALSE THEN
			a_pBufferZoneChildSIF[usiNumOfBufferZones-1]^.In.bolHangerDetected.intern := TRUE;
		END_IF
	ELSE
		fbSimulationTimer.IN := TRUE;
		a_pBufferZoneChildSIF[usiNumOfBufferZones-1]^.In.bolBufferFull.intern := FALSE;
	END_IF
			
	// bring hanger down to next stopperbuffer if top one is open
	ii:=usiNumOfBufferZones-1;
	WHILE ii>0 DO	
		IF ((a_pBufferZoneChildSIF[ii]^.Out.bolRetract.intern = TRUE) AND (abolRESimRetract[ii] = FALSE)) THEN
			IF (a_pBufferZoneChildSIF[ii]^.Cur.bolHangerDetected = TRUE) THEN
				a_pBufferZoneChildSIF[ii-1]^.In.bolBufferFull.intern := TRUE;
				abolRESimRetract[ii] := TRUE;
				IF a_pBufferZoneChildSIF[ii-1]^.Cfg.bolHasBufferFullSensor = FALSE THEN
					a_pBufferZoneChildSIF[ii-1]^.In.bolHangerDetected.intern := TRUE;
				END_IF
			END_IF
		ELSIF (a_pBufferZoneChildSIF[ii]^.Out.bolRetract.intern = FALSE) AND (abolRESimRetract[ii] = TRUE) THEN
			a_pBufferZoneChildSIF[ii-1]^.In.bolBufferFull.intern := FALSE;
			abolRESimRetract[ii] := FALSE;
		END_IF
		ii := ii - 1;
	END_WHILE			
END_IF
	
	


// Method refill all zones
CASE SubStateMachineRefill OF		
			
	// Check space in buffer X
	//-------------------------------
	0:
		// Check if number of hangers "per Pulse" have space in the next buffer
		// Condition: (zone[X].NumOfHangers + zone[ X + 1] .NumOfHangersPerPuls) < zone[X].MaxCapacity   			
(*		IF (((a_pBufferZoneChildSIF[intIndexRefill]^.Cur.dinNumOfHangersInBuffer + a_pBufferZoneChildSIF[intIndexRefill+1]^.Cfg.uinNumOfHangersPerPulse)
			< a_pBufferZoneChildSIF[intIndexRefill]^.Cfg.dinMaxCapacity) AND (a_pBufferZoneChildSIF[intIndexRefill+1]^.Cur.dinNumOfHangersInBuffer <> 0) AND (a_pBufferZoneChildSIF[intIndexRefill+1]^.Cur.bolHangerDetected = TRUE)) THEN
*)		IF ((a_pBufferZoneChildSIF[intIndexRefill]^.Cur.dinNumOfHangersInBuffer < a_pBufferZoneChildSIF[intIndexRefill]^.Cfg.dinMaxCapacity) AND 
			(a_pBufferZoneChildSIF[intIndexRefill+1]^.Cur.dinNumOfHangersInBuffer <> 0) AND (a_pBufferZoneChildSIF[intIndexRefill+1]^.Cur.bolHangerDetected = TRUE)) THEN
			
			// Send release command to buffer zone X+1
			a_pBufferZoneChildCIF[intIndexRefill+1]^.Job.intACmd:= STB_CmdState.cCMD_RELEASE;	
			SubStateMachineRefill:= 1;						
		ELSE
			// Check if a further zone exist?
			IF (intIndexRefill < (usiNumOfBufferZones-2)) THEN
				// Inc. index for next zone
				intIndexRefill:= intIndexRefill+1;
			ELSE
				// Restart at zone 1  
				intIndexRefill:= 0;
			END_IF
		END_IF
	
	// Check if zone X+1 is released
	//-------------------------------
	1:
		IF(a_pBufferZoneChildCIF[intIndexRefill+1]^.Job.intState = STB_CmdState.cSTA_RELEASE)THEN
			// Send stop command to buffer zone X+1
			a_pBufferZoneChildCIF[intIndexRefill+1]^.Job.intACmd:= cCMD_STOP;					
			SubStateMachineRefill:= 2;
			// Counter correction if no counter at inside of Buffer
			IF a_pBufferZoneChildSIF[intIndexRefill]^.Cfg.bolHasBufferFullSensor = FALSE THEN
				a_pBufferZoneChildSIF[intIndexRefill]^.Cur.dinNumOfHangersInBuffer := a_pBufferZoneChildSIF[intIndexRefill]^.Cur.dinNumOfHangersInBuffer + a_pBufferZoneChildSIF[intIndexRefill+1]^.Cfg.uinNumOfHangersPerPulse;
			END_IF
		END_IF	
	
	// Check if zone X+1 is stopped
	//-------------------------------
	2:
		IF(a_pBufferZoneChildCIF[intIndexRefill+1]^.Job.intState = cSTA_STOP)THEN
			udiTimeInStateRefill_ms:= 0;
			SubStateMachineRefill:= 3;					
		END_IF

	// Break
	//-------------------------------
	3:	
		// Increment time in state	
		udiTimeInStateRefill_ms:= udiTimeInStateRefill_ms + me.FUBInfo.udiSample_ms;
		IF (udiTimeInStateRefill_ms > SIf.Par.udiIntervalBufferFilling_ms) THEN
			// Back to first state
			SubStateMachineRefill:= 0;	
		END_IF
		
END_CASE
END_METHOD

METHOD RefillZones_parallel
VAR
	/// Loop variable
	ii: INT;
END_VAR
// Simulation
fbSimulationTimer.PT := UDINT_TO_TIME(SIf.Par.udiSimIncomingTime_ms);
IF (CIf.SwCfg.bolSimulation) THEN
	// Cyclicle input into the top stopperbuffer
	fbSimulationTimer(); // set time/reset timer
	IF fbSimulationTimer.Q = TRUE THEN
		fbSimulationTimer.IN := FALSE;
		a_pBufferZoneChildSIF[usiNumOfBufferZones-1]^.In.bolBufferFull.intern := TRUE;
		IF a_pBufferZoneChildSIF[usiNumOfBufferZones-1]^.Cfg.bolHasBufferFullSensor = FALSE THEN
			a_pBufferZoneChildSIF[usiNumOfBufferZones-1]^.In.bolHangerDetected.intern := TRUE;
		END_IF
	ELSE
		fbSimulationTimer.IN := TRUE;
		a_pBufferZoneChildSIF[usiNumOfBufferZones-1]^.In.bolBufferFull.intern := FALSE;
	END_IF
			
	// bring hanger down to next stopperbuffer if top one is open
	ii:=usiNumOfBufferZones-1;
	WHILE ii>0 DO	
		IF ((a_pBufferZoneChildSIF[ii]^.Out.bolRetract.intern = TRUE) AND (abolRESimRetract[ii] = FALSE)) THEN
			IF (a_pBufferZoneChildSIF[ii]^.Cur.bolHangerDetected = TRUE) THEN
				a_pBufferZoneChildSIF[ii-1]^.In.bolBufferFull.intern := TRUE;
				abolRESimRetract[ii] := TRUE;
				IF a_pBufferZoneChildSIF[ii-1]^.Cfg.bolHasBufferFullSensor = FALSE THEN
					a_pBufferZoneChildSIF[ii-1]^.In.bolHangerDetected.intern := TRUE;
				END_IF
			END_IF
		ELSIF (a_pBufferZoneChildSIF[ii]^.Out.bolRetract.intern = FALSE) AND (abolRESimRetract[ii] = TRUE) THEN
			a_pBufferZoneChildSIF[ii-1]^.In.bolBufferFull.intern := FALSE;
			abolRESimRetract[ii] := FALSE;
		END_IF
		ii := ii - 1;
	END_WHILE			
END_IF
	
	


// Method refill all zones
CASE SubStateMachineRefill OF		
			
	// Check space in buffer X
	//-------------------------------
	0:
		// Check if number of hangers "per Pulse" have space in the next buffer
		// Condition: (zone[X].NumOfHangers + zone[ X + 1] .NumOfHangersPerPuls) < zone[X].MaxCapacity   			
(*		IF (((a_pBufferZoneChildSIF[intIndexRefill]^.Cur.dinNumOfHangersInBuffer + a_pBufferZoneChildSIF[intIndexRefill+1]^.Cfg.uinNumOfHangersPerPulse)
			< a_pBufferZoneChildSIF[intIndexRefill]^.Cfg.dinMaxCapacity) AND (a_pBufferZoneChildSIF[intIndexRefill+1]^.Cur.dinNumOfHangersInBuffer <> 0) AND (a_pBufferZoneChildSIF[intIndexRefill+1]^.Cur.bolHangerDetected = TRUE)) THEN
*)		IF ((a_pBufferZoneChildSIF[intIndexRefill]^.Cur.dinNumOfHangersInBuffer < a_pBufferZoneChildSIF[intIndexRefill]^.Cfg.dinMaxCapacity) AND 
			(a_pBufferZoneChildSIF[intIndexRefill+1]^.Cur.dinNumOfHangersInBuffer <> 0) AND (a_pBufferZoneChildSIF[intIndexRefill+1]^.Cur.bolHangerDetected = TRUE))	
			
			AND (a_udiTimeInStateRefill_ms[intIndexRefill+1] > SIf.Par.udiIntervalBufferFilling_ms) THEN


		
			// Send release command to buffer zone X+1
			a_pBufferZoneChildCIF[intIndexRefill+1]^.Job.intACmd:= STB_CmdState.cCMD_RELEASE;	
			SubStateMachineRefill:= 1;						
		ELSE
			// Check if a further zone exist?
			IF (intIndexRefill < (usiNumOfBufferZones-2)) THEN
				// Inc. index for next zone
				intIndexRefill:= intIndexRefill+1;
			ELSE
				// Restart at zone 1  
				intIndexRefill:= 0;
			END_IF
		END_IF
	
	// Check if zone X+1 is released
	//-------------------------------
	1:
		IF(a_pBufferZoneChildCIF[intIndexRefill+1]^.Job.intState = STB_CmdState.cSTA_RELEASE)THEN
			// Send stop command to buffer zone X+1
			a_pBufferZoneChildCIF[intIndexRefill+1]^.Job.intACmd:= cCMD_STOP;					
			SubStateMachineRefill:= 2;
			// Counter correction if no counter at inside of Buffer
			IF a_pBufferZoneChildSIF[intIndexRefill]^.Cfg.bolHasBufferFullSensor = FALSE THEN
				a_pBufferZoneChildSIF[intIndexRefill]^.Cur.dinNumOfHangersInBuffer := a_pBufferZoneChildSIF[intIndexRefill]^.Cur.dinNumOfHangersInBuffer + a_pBufferZoneChildSIF[intIndexRefill+1]^.Cfg.uinNumOfHangersPerPulse;
			END_IF
		END_IF	
	
	// Check if zone X+1 is stopped
	//-------------------------------
	2:
		IF(a_pBufferZoneChildCIF[intIndexRefill+1]^.Job.intState = cSTA_STOP)THEN
			a_udiTimeInStateRefill_ms[intIndexRefill+1]:= 0;
			SubStateMachineRefill:= 3;					
		END_IF

	// Break
	//-------------------------------
	3:	
		// Increment time in state	
//		udiTimeInStateRefill_ms:= udiTimeInStateRefill_ms + me.FUBInfo.udiSample_ms;
//		IF (udiTimeInStateRefill_ms > SIf.Par.udiIntervalBufferFilling_ms) THEN
			// Back to first state
			SubStateMachineRefill:= 0;	
//		END_IF
		
END_CASE

// Increase time, if needed
FOR ii := 0 TO (usiNumOfBufferZones-1) DO
	a_udiTimeInStateRefill_ms[ii]:= a_udiTimeInStateRefill_ms[ii] + me.FUBInfo.udiSample_ms;
END_FOR
END_METHOD

METHOD PROTECTED sta_OFF : BOOL
// state implemetation
//--------------------------------------------------------------------------------------
// Entry action
	IF (me.StateMachine.intState<>me.StateMachine.intStateLastCycle) THEN
		me.StateMachine.intStateLastCycle := me.StateMachine.intState;
		;		
	END_IF

//--------------------------------------------------------------------------------------
// Cyclic action
	IF (me.StateMachine.intState=me.StateMachine.intStateLastCycle) THEN
		
		// Reset total counter
		SIf.Cur.dinHangersPassedTotal:= 0;
		
		// State Change Condition
		IF (me.Alarm.eActivAlmClass<>E_AlmClass.EOFF) AND (me.Alarm.eActivAlmClass<>E_AlmClass.OFF) THEN
			IF (me.intCmd=cCMD_STOP) THEN
				me.StateMachine.intStateNext := cSTA_STOPBusy;
			ELSIF (me.intCmd=cCMD_RUN) THEN 
				me.StateMachine.intStateNext := cSTA_RUNBusy;
			ELSIF(me.intCmd=SLB_CmdState.cCMD_RELEASE_ALL) THEN
				me.StateMachine.intStateNext := SLB_CmdState.cSTA_RELEASE_ALLBusy;
			END_IF
		END_IF
	END_IF


//--------------------------------------------------------------------------------------
// Exit action
	IF (me.StateMachine.intState<>me.StateMachine.intStateNext) THEN
		;
	END_IF
END_METHOD

METHOD PROTECTED sta_RELEASE_ALL : BOOL
// state implemetation
//--------------------------------------------------------------------------------------
// Entry action
	IF (me.StateMachine.intState<>me.StateMachine.intStateLastCycle) THEN
		me.StateMachine.intStateLastCycle := me.StateMachine.intState;	
		;
	END_IF

//--------------------------------------------------------------------------------------
// Cyclic action
	IF (me.StateMachine.intState=me.StateMachine.intStateLastCycle) THEN
		

		// State Change Condition
		IF ((me.intCmd=cCMD_STOP) OR (me.intCmd=cCMD_RUN)) THEN
			me.StateMachine.intStateNext := cSTA_STOPBusy;
		END_IF
	END_IF

//--------------------------------------------------------------------------------------
// Exit action
	IF (me.StateMachine.intState<>me.StateMachine.intStateNext) THEN
		;
	END_IF
END_METHOD

METHOD PROTECTED sta_RELEASE_ALLBusy : BOOL
// state implemetation
//--------------------------------------------------------------------------------------
// Entry action
	IF (me.StateMachine.intState<>me.StateMachine.intStateLastCycle) THEN
		me.StateMachine.intStateLastCycle := me.StateMachine.intState;
		
		bolAllZonesEmpty:= FALSE;
		
		// Init for refill sequence
		intIndexRefill:= 0;
		SubStateMachineRefill:=0;
	
		// Reset package counter
		SIf.Cur.dinHangersPassedPackage:= 0;
		dinPassedTotalZone1Old:= a_pBufferZoneChildSIF[0]^.Cur.dinHangersPassedTotal;
	
		// Initialize sub state machine
		me.SubStateMachine.intState:= cSTA_SUB_SEND_RELEASE; 
		me.SubStateMachine.intStateNext:= cSTA_SUB_SEND_RELEASE;
		
	END_IF

	
//--------------------------------------------------------------------------------------
// Cyclic action
	IF (me.StateMachine.intState=me.StateMachine.intStateLastCycle) THEN
		
		//--------------------------------------------------------------------------------------
		// This cyclic action runs until all buffer zones are emptied or job is stopped manually
		//--------------------------------------------------------------------------------------
			
		// Run this section until all zones are emptied
		IF NOT (THIS^.checkAllZonesEmpty()) THEN
			
			//----------------------------------------------------------------------
			// Continuous clocked emptying of buffer zone 1 (first zone, output)
			//----------------------------------------------------------------------		
			CASE me.SubStateMachine.intState OF	
				cSTA_SUB_WAIT_FOR_CMD:
					//..not used
			
				cSTA_SUB_SEND_RELEASE:				
					// Send release command to buffer zone 1
					a_pBufferZoneChildCIF[0]^.Job.intACmd:= STB_CmdState.cCMD_RELEASE;
								
					// State Change Condition
					IF(a_pBufferZoneChildCIF[0]^.Job.intState = STB_CmdState.cSTA_RELEASE)THEN
						me.SubStateMachine.intStateNext := cSTA_SUB_SEND_STOP;					
					END_IF		

				cSTA_SUB_SEND_STOP:
					// Send stop command to buffer zone 1
					a_pBufferZoneChildCIF[0]^.Job.intACmd:= cCMD_STOP;	
					
					// State Change Condition
					IF(a_pBufferZoneChildCIF[0]^.Job.intState = cSTA_STOP)THEN
						me.SubStateMachine.intStateNext := cSTA_SUB_BREAK;																
					END_IF	
			
				cSTA_SUB_BREAK:
					// Wait X-time and go back to state send release
					IF (me.SubStateMachine.udiTimeInState_ms > SIf.Par.udiIntervalBufferEmptying_ms) THEN
						me.SubStateMachine.intStateNext := cSTA_SUB_SEND_RELEASE;
					END_IF				
			END_CASE
					
			
			//----------------------------------------------------------------------
			// Continuous refill of all zones
			//----------------------------------------------------------------------
				
			// Only execute method if more than one buffer zones exist!
			// Note: Slide buffer controller can also used with only one buffer.
			IF ((usiNumOfBufferZones>1) AND (SIf.Cfg.bolRefill_parallel = FALSE)) THEN				
				THIS^.RefillZones();
			END_IF
			IF ((usiNumOfBufferZones>1) AND (SIf.Cfg.bolRefill_parallel = TRUE)) THEN				
				THIS^.RefillZones_parallel();
			END_IF			
		
		//-------------------------------		
		// All zones are emptied	
		//-------------------------------
		ELSE
			// send command STOP to all existing buffer zone child controller.
			THIS^.CmdToAllZones(cCMD_STOP);
			bolAllZonesEmpty:= TRUE;
		END_IF

		
		// Update package counter	
		IF (a_pBufferZoneChildSIF[0]^.Cur.dinHangersPassedTotal <> dinPassedTotalZone1Old) THEN
			// Calculate package counter dependent number of hangers per pulse in zone 1					
			SIf.Cur.dinHangersPassedPackage:= SIf.Cur.dinHangersPassedPackage + a_pBufferZoneChildSIF[0]^.Cfg.uinNumOfHangersPerPulse;			
		END_IF
		dinPassedTotalZone1Old:= a_pBufferZoneChildSIF[0]^.Cur.dinHangersPassedTotal;
		
		
		// State Change Condition
		IF (bolAllZonesEmpty=TRUE) THEN // All zones emptied -> RELEASE_ALL
			me.StateMachine.intStateNext := SLB_CmdState.cSTA_RELEASE_ALL;
		ELSIF(me.intCmd=cCMD_STOP) THEN
			me.StateMachine.intStateNext := cSTA_STOPBusy;		
		END_IF
		
	END_IF

//--------------------------------------------------------------------------------------
// Exit action
	IF (me.StateMachine.intState<>me.StateMachine.intStateNext) THEN
		;
	END_IF
END_METHOD

METHOD PROTECTED sta_RUN : BOOL
// state implemetation
//--------------------------------------------------------------------------------------
// Entry action
	IF (me.StateMachine.intState<>me.StateMachine.intStateLastCycle) THEN
		me.StateMachine.intStateLastCycle := me.StateMachine.intState;	
		;
	END_IF

//--------------------------------------------------------------------------------------
// Cyclic action
	IF (me.StateMachine.intState=me.StateMachine.intStateLastCycle) THEN
		
		//----------------------------------------------------------------------
		// Substates to let pass hanger(S) from zone 1
		// Triggered by command "Release" (common job interface)
		//----------------------------------------------------------------------		
		CASE me.SubStateMachine.intState OF	
			cSTA_SUB_WAIT_FOR_CMD:
				// Wait for command release
				IF (me.intCmd=STB_CmdState.cCMD_RELEASE) THEN
					CIf.Job.intACmd:=cSTA_DONE;
					me.SubStateMachine.intStateNext := cSTA_SUB_SEND_RELEASE;		
				END_IF
					
			cSTA_SUB_SEND_RELEASE:				
				// Send release command to buffer zone 1
				a_pBufferZoneChildCIF[0]^.Job.intACmd:= STB_CmdState.cCMD_RELEASE;
							
				// State Change Condition
				IF(a_pBufferZoneChildCIF[0]^.Job.intState = STB_CmdState.cSTA_RELEASE)THEN
					me.SubStateMachine.intStateNext := cSTA_SUB_SEND_STOP;					
				END_IF		

			cSTA_SUB_SEND_STOP:
				// Send stop command to buffer zone 1
				a_pBufferZoneChildCIF[0]^.Job.intACmd:= cCMD_STOP;	
				
				// State Change Condition
				IF(a_pBufferZoneChildCIF[0]^.Job.intState = cSTA_STOP)THEN
					me.SubStateMachine.intStateNext := cSTA_SUB_WAIT_FOR_CMD;																
				END_IF	
		
			cSTA_SUB_BREAK:
				//..not used	
		
		END_CASE
				
		
		//----------------------------------------------------------------------
		// Continuous refill of all zones
		//----------------------------------------------------------------------
		
		// Only execute method if more than one buffer zones exist!
		// Note: Slide buffer controller can also used with only one buffer.
		IF ((usiNumOfBufferZones>1) AND (SIf.Cfg.bolRefill_parallel = FALSE)) THEN				
			THIS^.RefillZones();
		END_IF
		IF ((usiNumOfBufferZones>1) AND (SIf.Cfg.bolRefill_parallel = TRUE)) THEN				
			THIS^.RefillZones_parallel();
		END_IF
			
			
		// Sub state machine general handling
		me.SubStateMachine.intStateLastCycle := me.SubStateMachine.intState;
		CIf.Job.strSubState := THIS^.getCmdState(intCmdState:=me.SubStateMachine.intState,bolState:=TRUE);
		IF (me.SubStateMachine.intState<>me.SubStateMachine.intStateNext) THEN
			me.SubStateMachine.intState := me.SubStateMachine.intStateNext;  // set next state for next cycle
			me.SubStateMachine.udiTimeInState_ms := 0; // reset timer
			// log state change -> open point
		ELSE
			// increment time in state	
			me.SubStateMachine.udiTimeInState_ms := me.SubStateMachine.udiTimeInState_ms + me.FUBInfo.udiSample_ms;
		END_IF
	
		
		// State Change Condition
		IF ((me.intCmd=cCMD_STOP) AND (me.SubStateMachine.intState=cSTA_SUB_WAIT_FOR_CMD))THEN
			me.StateMachine.intStateNext := cSTA_STOPBusy;
		ELSIF ((me.intCmd=STB_CmdState.cCMD_RELEASE_ALL) AND (me.SubStateMachine.intState=cSTA_SUB_WAIT_FOR_CMD))THEN
			me.StateMachine.intStateNext := STB_CmdState.cSTA_RELEASE_ALLBusy;
		END_IF
	END_IF

//--------------------------------------------------------------------------------------
// Exit action
	IF (me.StateMachine.intState<>me.StateMachine.intStateNext) THEN
		;
	END_IF
END_METHOD

METHOD PROTECTED sta_RUNBusy : BOOL
// state implemetation
//--------------------------------------------------------------------------------------
// Entry action
	IF (me.StateMachine.intState<>me.StateMachine.intStateLastCycle) THEN
		me.StateMachine.intStateLastCycle := me.StateMachine.intState;
		
		// Init for refill sequence
		intIndexRefill:= 0;
		SubStateMachineRefill:=0;
	
		// Initialize sub state machine
		me.SubStateMachine.intState:= cSTA_SUB_WAIT_FOR_CMD; 
		me.SubStateMachine.intStateNext := cSTA_SUB_WAIT_FOR_CMD;
	END_IF

	
//--------------------------------------------------------------------------------------
// Cyclic action
	IF (me.StateMachine.intState=me.StateMachine.intStateLastCycle) THEN
			
	
		// State Change Condition	
		IF (TRUE) THEN
			me.StateMachine.intStateNext := cSTA_RUN;		
		END_IF

	END_IF

//--------------------------------------------------------------------------------------
// Exit action
	IF (me.StateMachine.intState<>me.StateMachine.intStateNext) THEN
		;
	END_IF
END_METHOD

METHOD PROTECTED sta_STOP : BOOL
// state implemetation
//--------------------------------------------------------------------------------------
// Entry action
	IF (me.StateMachine.intState<>me.StateMachine.intStateLastCycle) THEN
		me.StateMachine.intStateLastCycle := me.StateMachine.intState;
		;
	END_IF

//--------------------------------------------------------------------------------------
// Cyclic action
	IF (me.StateMachine.intState=me.StateMachine.intStateLastCycle) THEN

	
		// State Change Condition	
		IF (me.intCmd = cCMD_RUN) THEN 
			me.StateMachine.intStateNext := cSTA_RUNBusy;
		ELSIF(me.intCmd = SLB_CmdState.cCMD_RELEASE_ALL) THEN
			me.StateMachine.intStateNext := SLB_CmdState.cSTA_RELEASE_ALLBusy;
		END_IF
	END_IF

//-------------------------------------------------------------------------------------
// Exit action
	IF (me.StateMachine.intState<>me.StateMachine.intStateNext) THEN
		;
	END_IF
END_METHOD

METHOD PROTECTED sta_STOPBusy : BOOL
// state implemetation
//--------------------------------------------------------------------------------------
// Entry action
	IF (me.StateMachine.intState<>me.StateMachine.intStateLastCycle) THEN
		me.StateMachine.intStateLastCycle := me.StateMachine.intState;
		
		// send command STOP to all existing buffer zone child controller.
		THIS^.CmdToAllZones(cCMD_STOP);

	END_IF

//--------------------------------------------------------------------------------------
// Cyclic action
	IF (me.StateMachine.intState=me.StateMachine.intStateLastCycle) THEN
			
				
		// State Change Condition
		// Check if all STOPPED
		IF (THIS^.checkStateAllZones(cSTA_STOP)) THEN
			me.StateMachine.intStateNext := cSTA_STOP;
		END_IF
	END_IF

//--------------------------------------------------------------------------------------
// Exit action
	IF (me.StateMachine.intState<>me.StateMachine.intStateNext) THEN
		;
	END_IF
END_METHOD

METHOD PROTECTED StateMachine : BOOL
SUPER^.StateMachine();

// main statemachine of base controller
CASE me.StateMachine.intState OF
    cSTA_STOPBusy: 
        THIS^.sta_STOPBusy();
    cSTA_STOP: 
        THIS^.sta_STOP();
	cSTA_RUNBusy: 
        THIS^.sta_RUNBusy();
    cSTA_RUN: 
        THIS^.sta_RUN();				
    SLB_CmdState.cSTA_RELEASE_ALLBusy: 
        THIS^.sta_RELEASE_ALLBusy();
    SLB_CmdState.cSTA_RELEASE_ALL: 
        THIS^.sta_RELEASE_ALL();
END_CASE;
END_METHOD

END_FUNCTION_BLOCK

// POUs/Controller/Lvl1/DPJ (DecisionPoint Junction)/FB_DPJ
FUNCTION_BLOCK FB_DPJ EXTENDS FB_CtrlBase
VAR_INPUT
	/// Sensor Counter into the system
	In_bolCounterIn: BOOL;
	/// Sensor Counter out of the system
	In_bolCounterOut: BOOL;
	/// Hanger exactly at RFID Position
	In_bolHangerDetector: BOOL;
	///pointer to function block RFID Reader
	p_fbRFW: POINTER TO FB_RFW;
END_VAR
VAR
	/// Specific interface struct for public access
	SIf: T_Ctrl_SIf_DPJ;
	/// Interface to Childs
	pRFW_CIF: POINTER TO T_Ctrl_CIf;
	pRFW_SIF: POINTER TO T_Ctrl_SIf_RFW;
	/// Childs of Junctions
	/// List of pointers to Childs
	a_pMultiChildCtrl: ARRAY[0..Base_Const.cMaxNrOfChilds] OF POINTER TO FB_JUN;
	/// List of childs common interface
	a_pMultiChildCIF: ARRAY[0..Base_Const.cMaxNrOfChilds] OF POINTER TO T_Ctrl_CIf;
	/// List of childs specific interface for additional parameters or cur
	a_pMultiChildSIF: ARRAY[0..Base_Const.cMaxNrOfChilds] OF POINTER TO T_Ctrl_SIf_JUN;
	usiNumOfMultiChild: USINT;
	usiNumOfValidPointerMultiChild: USINT;
	/// Hashtable
	aTblDecision: ARRAY[0..cintMaxDecisions] OF T_DecisionElement;
	/// Datachannel
	/// Internal Variable Data Channel Variables
	intStatemachine: INT;
	/// Data not correct
	bolDataBad: BOOL;
	/// Data found
	bolDataFound: BOOL;
	/// Retry Counts for error message
	intCountRetry: INT;
	/// Data Channel Specific Variable
	intIndexOldest: INT;
	/// Date and time of the oldes imput
	dtOldestTag: DT;
	/// Datachannel to send done job
	fbDtChnToLine_JobDone: FB_DtChnToLine_JobDone;
	/// Error information from Job Done
	intStateDtChnToLine_JobDone: INT;
	/// Internal Variable
	dtActualTime: DT;
	/// Actual Time and date
	dtDeleteTime: DT;
	/// New RFID Tag ID Job found and actualisised in Hashtable
	bolJobFound: BOOL;
	/// Rising Edge detection of Hanger at RFID Position
	bolREHangerDetection: BOOL;
	/// Rising Edge detection of Hanger Counter input
	bolRECounterIn: BOOL;
	/// Rising Edge detection of Hanger Counter output
	bolRECounterOut: BOOL;
	/// No Job active
	bolNoJobActive: BOOL;
	/// Last RFID Tag ID
	uliRFID_Tag_old: ULINT;
	/// Loop variable for RFID check
	uinLoopRFID: UINT;
	/// Transportposition from last cycle
	dinTransportPosition_old_um: DINT;
	/// Driven Way from last to actual cycle
	dinTransportDifferenz_um: DINT;
	/// Actual position of the hanger at the RFID Reader
	dinPositionRFID_um: DINT;
	/// Index of the actual hanger at RFID Position 
	intIndexActualHanger: INT;
	/// Index of the RFID 
	intIndexActualRFID: INT;
	/// Loop Variable
	intI: INT;
	/// Table for line control data channel simulation
	aSimDataChlLine: ARRAY[0..cintMaxDecisions] OF T_SimDtChn;
	/// State for simulation data channel to PLC
	intSimStateChlToPLC: INT;
	/// State for simulation data channel to Line
	intSimStateChlToLine: INT;
	intIndexSetEntry: INT;
	intIndexGetEntry: INT;
	dinSimTimerAcknowledge: DINT;
	dinSimTimerProcessTimeLine: DINT;
	// Time for waiting for the second signal (Sensor or RFID) 
	udiWaitingForSecondSignal_ms: UDINT;
END_VAR
VAR CONSTANT
	cSTA_SUB_SimWaitForDataReady: INT := 1000;
	cSTA_SUB_SimAcknowledgeFromLine: INT := 1001;
	cSTA_SUB_SimWaitForNewData: INT := 1002;
	cSTA_SUB_SimProcessingTimeOnLineControl: INT := 1003;
	cSTA_SUB_SimNewJobForPLC: INT := 1004;
	cSTA_SUB_SimGetData: INT := 1005;
	cSTA_SUB_SimWaitJobDone: INT := 1006;
	cSimDataState_DONE: INT := -1;
	cSimDataState_Ready: INT := 1;
	cSimDataState_Retry: INT := -99;
END_VAR

(*__________________________________________________________________________________________________
¦	
¦	Vistaprint Schweiz GmbH
¦	CH - 8401 Winterthur
¦
¦	www.vistaprint.ch - info@vistaprint.ch
¦___________________________________________________________________________________________________

Function desription:
Desictionpoint and Junction parent
This controller communicate with a datachannel to the Linecontroller to get the hashtable
With a RFID Child it reads every tag and controlls the junctions to open the correct one


History:
Version		Date			Author		Comment
---------------------------------------------------------------------------------------------------
0.00.1		23.08.2013		AVM/PRE		Start history
0.00.2		02.10.2013		VP/RE		Skip zero entries in hash table. Fixed junction number count (was not set after init). Fixed data validation in DataChannel->cSTA_SUB_Data_CheckData.
0.00.3		04.10.2013		AVM/DSC		Changed timestamp element in data channel structure from DT to String
0.00.4		30.10.2013		AVM/DSC		Change request from REN (15.10.2013). Now it's possible to send a new job also if a hanger is on the way to a junction.
										Add. modifications in method "DtChnToPLC_Decision" for states DELETE_ALL, DELETE_JUNCTION and DELETE_ID after tests together with line control.				
0.00.5		09.12.2013		AVME/DSC	Modification in method "checkStateAllMultiChild".
										Special condition: In case if the child is in state ERROR and STOP is requested. Set child as checked.
										Parent controller need state STOP that automatic stop sequence can work for all other childs.
0.00.6		22.10.2014		AVME/MRU	New settings (SIf.Par.udiTimeMaxJob_s := 60; cintMaxDecisions: INT := 100;)
										Reworked in sta_STOPBusy calculation of bolNoJobActive
0.00.7		03.02.2014		AVME/MRU	sta_RUN entry action reworked
0.00.8		24.04.2014		AVME/MRU	Replaced with latest version of ShirtStream
0.00.9		10.07.2014		AVME/MRU	Check Time-Out Waitung for Signal or RFID-Tag, new function for preventing miss-readed Tags (so called N+1-Problem)
0.00.10		16.07.2014		AVME/MRU	Some Bugs fixed
										
___________________________________________________________________________________________________*)


IF (me.bolActivate)  AND (p_fbRFW<>0) AND (THIS^.checkChildPointer()) THEN // cyclic call enabled
	IF (CIf.Info.bolInitDone=FALSE) THEN // first cycle -> init
		CtrlInit();
		CIf.Info.bolInitDone := TRUE;
	ELSE
		CycleStartDuty();
	
		Always();
		
		StateMachine();
		
		CycleEndDuty();
	END_IF
END_IF;

METHOD AddJunction
VAR_INPUT
	p_MultiChild: POINTER TO FB_JUN;
END_VAR

// Method add the pointer address of the buffer zone child controller to the array list.
IF (usiNumOfMultiChild <= (Base_Const.cMaxNrOfChilds-1)) THEN
	// Add buffer zone child controller to list
	a_pMultiChildCtrl[usiNumOfMultiChild] := p_MultiChild;
	// Inc. number of buffer zones
	usiNumOfMultiChild:= usiNumOfMultiChild+1;
	// Check if the pointer is valid
	IF (p_MultiChild<>0) THEN
		usiNumOfValidPointerMultiChild:= usiNumOfValidPointerMultiChild+1;
	END_IF
END_IF
END_METHOD

METHOD PROTECTED Always : BOOL
VAR
	fbGetSystemTime: GETSYSTEMTIME;
	stfileTime: T_FILETIME;
	intI: INT;
	ii: INT;
END_VAR
IF (me.bolChangeBackToAUTO=TRUE) THEN // switch mode to automatic switch off controller
	//me.StateMachine.intStateNext := cSTA_OFFBusy;
	//me.bolChangeBackToAUTO := FALSE; // for cylinder no change to off when switch to automatic!!
END_IF

SUPER^.Always();

// ---------------------------------------------------------------------------------
// check child me and set parent alarm class
checkChildAlmClass();

// ----------------------------------------------------------------------------------
// SIMULATION OF LINE CONTROL DATA CHANNEL
// ----------------------------------------------------------------------------------

IF (SIf.Cfg.bolSimDtChLine) THEN

	// STATE MACHINE FOR SIMULATION DATA CHANNEL TO LINE
	CASE intSimStateChlToLine OF
		
		cSTA_SUB_SimGetData:
			// Set Acknowledge from line
			pRFW_SIF^.DtChnToLine.stNewRfid.intDataState:= cSimDataState_DONE;
			intSimStateChlToLine:= cSTA_SUB_SimWaitForDataReady;
			
		cSTA_SUB_SimWaitForDataReady:
			// Look at the RFW instance! Wait for new RFID 			
			IF (pRFW_SIF^.DtChnToLine.stNewRfid.intDataState = cSimDataState_Ready) THEN
				// Ring buffer handling
				IF (intIndexSetEntry > cintMaxDecisions) THEN
					// Start at zero, override entries
					intIndexSetEntry:= 0;
				END_IF
				// Copy data to sim data channel buffer
				aSimDataChlLine[intIndexSetEntry].stDecision.uliRFID:= pRFW_SIF^.DtChnToLine.stNewRfid.uliTagID;
				aSimDataChlLine[intIndexSetEntry].stDecision.strID:= pRFW_SIF^.DtChnToLine.stNewRfid.strID;
				aSimDataChlLine[intIndexSetEntry].strTimestamp:= pRFW_SIF^.DtChnToLine.stNewRfid.strTimestamp;
				aSimDataChlLine[intIndexSetEntry].intDataState:= pRFW_SIF^.DtChnToLine.stNewRfid.intDataState;
		
				dinSimTimerAcknowledge:= SIf.Par.dinSimTimeAcknowledgeDataChl_ms;
				intSimStateChlToLine:= cSTA_SUB_SimAcknowledgeFromLine;
			END_IF
		
		cSTA_SUB_SimAcknowledgeFromLine:
			// Wait X-time
			IF (dinSimTimerAcknowledge <= 0) THEN			 
				aSimDataChlLine[intIndexSetEntry].intInternalSimState:= 1; //1=SimDataPLCToLineDone
				intIndexSetEntry:= intIndexSetEntry + 1;
				// Set Acknowledge from line, line has received new RFID
				//pRFW_SIF^.DtChnToLine.stNewRfid.intDataState:= cSimDataState_DONE;
				intSimStateChlToLine:= cSTA_SUB_SimGetData;
			END_IF	

	(*
		cSTA_SUB_SimWaitForDataReady:
			// Wait for new data from channel to line
			IF (SIf.DtChnToLine.stJobDone.intDataState = cSimDataState_Ready) THEN
				// Ring buffer handling
				IF (intIndexSetEntry > cintMaxDecisions) THEN
					// Start at zero, override entries
					intIndexSetEntry:= 0;
				END_IF
				// Copy data to sim data channel buffer
				aSimDataChlLine[intIndexSetEntry].stDecision.uliRFID:= SIf.DtChnToLine.stJobDone.stDecision.uliRFID;
				aSimDataChlLine[intIndexSetEntry].stDecision.strID:= SIf.DtChnToLine.stJobDone.stDecision.strID;
				aSimDataChlLine[intIndexSetEntry].strTimestamp:= SIf.DtChnToLine.stJobDone.strTimestamp;
				aSimDataChlLine[intIndexSetEntry].intDataState:= SIf.DtChnToLine.stJobDone.intDataState;
		
				dinSimTimerAcknowledge:= SIf.Par.dinSimTimeAcknowledgeDataChl_ms;
				intSimStateChlToLine:= cSTA_SUB_SimAcknowledgeFromLine;
			END_IF
		
		cSTA_SUB_SimAcknowledgeFromLine:
			// Wait X-time
			IF (dinSimTimerAcknowledge <= 0) THEN			 
				aSimDataChlLine[intIndexSetEntry].intInternalSimState:= 1; //1=SimDataPLCToLineDone
				intIndexSetEntry:= intIndexSetEntry + 1;
				// Set Acknowledge from line, line has received new RFID
				SIf.DtChnToLine.stJobDone.intDataState:= cSimDataState_DONE;
				intSimStateChlToLine:= cSTA_SUB_SimWaitForDataReady;
			END_IF
	 *)
	END_CASE
			
	// Timer handling outside of state machine
	IF (dinSimTimerAcknowledge > 0) THEN
		dinSimTimerAcknowledge:= dinSimTimerAcknowledge - UDINT_TO_DINT(me.FUBInfo.udiSample_ms);
	END_IF
			
		
	// STATE MACHINE FOR SIMULATION DATA CHANNEL TO PLC
	CASE intSimStateChlToPLC OF
	
		cSTA_SUB_SimWaitForNewData:
			// If data channel is enabled
			IF (Sif.Cfg.bolSimEnableDtChToPLC) THEN		
				// Ring buffer handling
				IF (intIndexGetEntry > cintMaxDecisions) THEN
					// Start at zero, override entries
					intIndexGetEntry:= 0;
				END_IF	
				// Simulation Data To Line Done?
				IF (aSimDataChlLine[intIndexGetEntry].intInternalSimState = 1) THEN
					// Simulation line to PLC in work
					aSimDataChlLine[intIndexGetEntry].intInternalSimState:= 2;  //2=SimDataLineToPLCInWork
					dinSimTimerProcessTimeLine:= SIf.Par.dinSimProcessTimeOnLineCtrl_ms;
					intSimStateChlToPLC:= cSTA_SUB_SimProcessingTimeOnLineControl;			
				END_IF
			END_IF
			
		cSTA_SUB_SimProcessingTimeOnLineControl:
			// Wait X-time
			IF (dinSimTimerProcessTimeLine <= 0) THEN			 
				intSimStateChlToPLC:= cSTA_SUB_SimNewJobForPLC;
			END_IF
			
		cSTA_SUB_SimNewJobForPLC:

			// NEW Job data 
			// RFID
			SIf.DtChnToPLC.stNewDecision.stDecision.uliRFID:= aSimDataChlLine[intIndexGetEntry].stDecision.uliRFID;
			// Define the Target -> Which Junction?
			SIf.DtChnToPLC.stNewDecision.stDecision.dinTarget:= SIf.Par.dinSimTarget;	
			
			// Set info to data channel: New data arrived -> set JOB CMD "NEW"
			SIf.DtChnToPLC.stNewDecision.intDataState:= cSimDataState_Ready;
			SIf.DtChnToPLC.stNewDecision.intJob:= E_Decision_Job.NEW;		
			// Next step
			intSimStateChlToPLC:= cSTA_SUB_SimWaitJobDone;
			
		cSTA_SUB_SimWaitJobDone:
			// Retry
			IF (SIf.DtChnToPLC.stNewDecision.intDataState = cSimDataState_Retry) THEN
 				// Retry step
				intSimStateChlToPLC:= cSTA_SUB_SimNewJobForPLC;	
			END_IF
			// Done
			IF (SIf.DtChnToPLC.stNewDecision.intDataState = cSimDataState_DONE) THEN
				aSimDataChlLine[intIndexGetEntry].intInternalSimState:= 0;
				//aSimDataChlLine[intIndexGetEntry].stDecision.uliRFID:=0;
				//aSimDataChlLine[intIndexGetEntry].stDecision.dinTarget:=0;
				//aSimDataChlLine[intIndexGetEntry].stDecision.strID:='';
				
				// Get Next entry
				IF (SIf.Par.intSimDischargingEveryXtenHanger = 1) THEN
					intIndexGetEntry:=intIndexGetEntry + 1;
				ELSE
					// Calculate, which one is the next?
					IF ((intIndexGetEntry + SIf.Par.intSimDischargingEveryXtenHanger) <= cintMaxDecisions) THEN
						intIndexGetEntry:= intIndexGetEntry + SIf.Par.intSimDischargingEveryXtenHanger;
					ELSE
						// Correction of index
						intIndexGetEntry:= (intIndexGetEntry + SIf.Par.intSimDischargingEveryXtenHanger) - cintMaxDecisions - 1;
					END_IF					
				END_IF				
				// Next step
				intSimStateChlToPLC:= cSTA_SUB_SimWaitForNewData;		
			END_IF	
	END_CASE	
	
	// Timer handling outside of state machine
	IF (dinSimTimerProcessTimeLine > 0) THEN
		dinSimTimerProcessTimeLine:= dinSimTimerProcessTimeLine - UDINT_TO_DINT(me.FUBInfo.udiSample_ms);
	END_IF	
		
	
//Simulation disabled
ELSE
	// Set init states
	intSimStateChlToLine:= cSTA_SUB_SimGetData;
	intSimStateChlToPLC:= cSTA_SUB_SimWaitForNewData;
	
	intIndexSetEntry:=0;
	intIndexGetEntry:=0;
END_IF
// ----------------------------------------------------------------------------------
// SIMULATION OF LINE CONTROL DATA CHANNEL
// ----------------------------------------------------------------------------------

// ----------------------------------------------------------------------------------
// cyclic actions outside of statemachine
fbGetSystemTime(timeLoDW=>stfileTime.dwLowDateTime, timeHiDW=>stfileTime.dwHighDateTime);
dtActualTime := FILETIME_TO_DT( stfileTime );
dtDeleteTime := DINT_TO_DT(DT_TO_DINT(dtActualTime) - UDINT_TO_DINT(SIf.Par.udiTimeMaxJob_s));	

// Cyclicel Hashtable work
FOR intI:=0 TO cintMaxDecisions DO

	// Delete old jobs by time 	
	IF  (aTblDecision[intI].dtTimeJob < dtDeleteTime) THEN
		IF aTblDecision[intI].eState = E_DecisionState.Finished THEN			
			// Delete done job
			aTblDecision[intI].eState := 0;
			aTblDecision[intI].dinActPos_um := 0;
			aTblDecision[intI].dtTimeJob := DINT_TO_DT(0);
			aTblDecision[intI].dtTimeRFID := DINT_TO_DT(0);
			aTblDecision[intI].stDecision.dinTarget := 0;
			aTblDecision[intI].stDecision.uliRFID := 0;
			aTblDecision[intI].stDecision.strID := '';
		ELSIF aTblDecision[intI].eState = E_DecisionState.Wait THEN
			// Job not startet, set error
			// Set Alarm: SIf.Alm[4].strText := 'Job Timeout, delete Job';
			pfbAlarmCtrl^.setAlarm(CIf.Info.intCtrlId,4,intI,ADR(SIf.Alm),E_AlmState.RST,CIf.Job.eMe_ActivAlmClass);
			// Clear Job										
			aTblDecision[intI].eState := E_DecisionState.none;
			aTblDecision[intI].dinActPos_um := 0;
			aTblDecision[intI].dtTimeJob := DINT_TO_DT(0);
			aTblDecision[intI].dtTimeRFID := DINT_TO_DT(0);
			aTblDecision[intI].stDecision.dinTarget := 0;
			aTblDecision[intI].stDecision.uliRFID := 0;
			aTblDecision[intI].stDecision.strID := '';	
		ELSIF (aTblDecision[intI].eState = E_DecisionState.DriveOut OR aTblDecision[intI].eState = E_DecisionState.Processed) THEN // MRU 17.07.2014 added
			// Drive Out Acknowledge missing, set error
			// Set Alarm: SIf.Alm[15].strText := 'Drive Out Acknowledge missing, delete Job';
			pfbAlarmCtrl^.setAlarm(CIf.Info.intCtrlId,15,intI,ADR(SIf.Alm),E_AlmState.RST,CIf.Job.eMe_ActivAlmClass);
			// Clear Job										
			aTblDecision[intI].eState := E_DecisionState.none;
			aTblDecision[intI].dinActPos_um := 0;
			aTblDecision[intI].dtTimeJob := DINT_TO_DT(0);
			aTblDecision[intI].dtTimeRFID := DINT_TO_DT(0);
			aTblDecision[intI].stDecision.dinTarget := 0;
			aTblDecision[intI].stDecision.uliRFID := 0;
			aTblDecision[intI].stDecision.strID := '';				
		END_IF
	END_IF
	
	
	// Delete jobs where the hanger crossed the last junction but did not get a target number assigned by line control.
	IF ((aTblDecision[intI].dinActPos_um > (SIf.Cur.dinDistanceToFarthestJunction + SIf.Par.dinDistanceOffsetUntilDelJob_um)) AND (aTblDecision[intI].stDecision.dinTarget <= 0)) THEN
		IF (aTblDecision[intI].eState = E_DecisionState.WayToJunction) THEN			
			aTblDecision[intI].eState := 0;
			aTblDecision[intI].dinActPos_um := 0;
			aTblDecision[intI].dtTimeJob := DINT_TO_DT(0);
			aTblDecision[intI].dtTimeRFID := DINT_TO_DT(0);
			aTblDecision[intI].stDecision.dinTarget := 0;
			aTblDecision[intI].stDecision.uliRFID := 0;
			aTblDecision[intI].stDecision.strID := '';	
		END_IF
	END_IF

	// Write an Error when the hanger crossed the last junction but did not get finished
	IF ((aTblDecision[intI].dinActPos_um > (SIf.Cur.dinDistanceToFarthestJunction + SIf.Par.dinDistanceOffsetUntilDelJob_um)) AND (aTblDecision[intI].stDecision.dinTarget > 0)) THEN
		IF (aTblDecision[intI].eState = E_DecisionState.WayToJunction) THEN			
			IF (SIf.Cfg.bolStopAtPassLastJunction = TRUE) THEN	// E_AlmClass.STOP
				// SIf.Alm[13].strText := 'Hanger passed the last instead of selected junction';
				pfbAlarmCtrl^.setAlarm(CIf.Info.intCtrlId,13,0,ADR(SIf.Alm),E_AlmState.RST,CIf.Job.eMe_ActivAlmClass);
			ELSE // E_AlmClass.INFO
				// SIf.Alm[12].strText := 'Hanger passed the last instead of selected junction';
				pfbAlarmCtrl^.setAlarm(CIf.Info.intCtrlId,12,0,ADR(SIf.Alm),E_AlmState.RST,CIf.Job.eMe_ActivAlmClass);
			END_IF
			aTblDecision[intI].eState := 0;
			aTblDecision[intI].dinActPos_um := 0;
			aTblDecision[intI].dtTimeJob := DINT_TO_DT(0);
			aTblDecision[intI].dtTimeRFID := DINT_TO_DT(0);
			aTblDecision[intI].stDecision.dinTarget := 0;
			aTblDecision[intI].stDecision.uliRFID := 0;
			aTblDecision[intI].stDecision.strID := '';	
		END_IF
	END_IF
	
	// Check if a hanger passed the junction to send a message to line
	IF (aTblDecision[intI].eState = E_DecisionState.DriveOut) THEN
		IF (SIf.Cfg.bolDtChToLine_send = TRUE) THEN			
			IF fbDtChnToLine_JobDone.Creat(In_strTimestamp:= DT_TO_STRING(dtActualTime),In_stDecision := aTblDecision[intI].stDecision,) = 1 THEN
				IF SIf.Cur.dinCurrentItemCount > 0 THEN
					SIf.Cur.dinCurrentItemCount := SIf.Cur.dinCurrentItemCount - 1;
				END_IF
				aTblDecision[intI].eState := E_DecisionState.Finished;
			ELSE	
				IF NOT (SIf.cfg.bolSimDtChLine) THEN						
					// Set Alarm: SIf.Alm[9].strText := 'Data Channel Error Send Data';
					pfbAlarmCtrl^.setAlarm(CIf.Info.intCtrlId,9,0,ADR(SIf.Alm),E_AlmState.RST,CIf.Job.eMe_ActivAlmClass);
				ELSE
					// MRU 16.7.2014: Added to clean up Table in Simulation
					aTblDecision[intI].eState := E_DecisionState.Finished;
				END_IF
			END_IF
		ELSE
			IF SIf.Cur.dinCurrentItemCount > 0 THEN
				SIf.Cur.dinCurrentItemCount := SIf.Cur.dinCurrentItemCount - 1;
			END_IF
			aTblDecision[intI].eState := E_DecisionState.Finished;
		END_IF
	END_IF	

END_FOR

// Count Hangers in Controller
// Hanger In
IF SIf.In.bolCounterIn.intern = TRUE AND bolRECounterIn = FALSE THEN
	bolRECounterIn := TRUE;
	SIf.Cur.dinCurrentItemCount := SIf.Cur.dinCurrentItemCount + 1;
ELSIF SIf.In.bolCounterIn.intern = FALSE THEN
	bolRECounterIn := FALSE;
END_IF
// Hanger Out
IF SIf.In.bolCounterOut.intern = TRUE AND bolRECounterOut = FALSE THEN
	bolRECounterOut := TRUE;
	IF SIf.Cur.dinCurrentItemCount > 0 THEN
		SIf.Cur.dinCurrentItemCount := SIf.Cur.dinCurrentItemCount - 1;
	END_IF
ELSIF SIf.In.bolCounterOut.intern = FALSE THEN
	bolRECounterOut := FALSE;
END_IF

// Current Value Mapping internal
SIf.Cur.dinMaxCapacity := SIf.Cfg.dinMaxCapacity;
SIf.Cfg.intCountJunctions := usiNumOfMultiChild;

// Current Value Mapping to Childs
FOR ii:=0 TO usiNumOfMultiChild-1 BY 1 DO	
	a_pMultiChildSIF[ii]^.Cur.dinTransportPosition_um := SIf.Cur.dinTransportPosition_um;
	a_pMultiChildSIF[ii]^.Cur.dinTransportspeed_um_s := SIf.Cur.dinTransportspeed_um_s;

END_FOR

IF (me.StateMachine.intState<>cSTA_SINGLE_ANSWER) THEN
	// Communication to the Line Controll over Data Channel
	THIS^.DtChnToPLC_Decision();
	fbDtChnToLine_JobDone.bolResetError := CIf.Job.bolAlmReset;
	fbDtChnToLine_JobDone.pSIf := ADR(SIf);
	fbDtChnToLine_JobDone();
	IF fbDtChnToLine_JobDone.intError <> 0 THEN
		// Set Alarm: SIf.Alm[9].strText := 'Data Channel Error Send Data';
		pfbAlarmCtrl^.setAlarm(CIf.Info.intCtrlId,9,fbDtChnToLine_JobDone.intError,ADR(SIf.Alm),E_AlmState.RST,CIf.Job.eMe_ActivAlmClass);	
	END_IF
END_IF

// ----------------------------------------------------------------------------------
// Conditions Always
// overrule error always from base -> no EOFF State!! in EOFF go to OFF
IF (me.StateMachine.intStateNext = cSTA_EOFFBusy) THEN
	IF (me.StateMachine.intState=cSTA_OFF) THEN
		me.StateMachine.intStateNext := cSTA_OFF;
	ELSE // stay in OFF
		me.StateMachine.intStateNext := cSTA_OFFBusy;
	END_IF
END_IF
END_METHOD

METHOD PROTECTED checkAlmClassAllMultiChild : BOOL
VAR_INPUT
	In_AlmClass: E_AlmClass;
END_VAR
VAR
	ii: INT;
END_VAR
// Method check the current alm class of all zones and give back 
// TRUE if one of the childs corresponds the input "In_AlmClass" of this method 

//Init
checkAlmClassAllMultiChild:= FALSE;

// Loop over all childs
FOR ii:=0 TO usiNumOfMultiChild-1 BY 1 DO
	// Check about active alm class	
	IF (a_pMultiChildCIF[ii]^.Job.eMe_ActivAlmClass = In_AlmClass) THEN
		checkAlmClassAllMultiChild:= TRUE;
	END_IF
END_FOR
END_METHOD

METHOD checkChildAlmClass : BOOL
//------------------------------------------------------------------------------------------------------
// check child alarm classes
IF (pRFW_CIF^.Job.eMe_ActivAlmClass=E_AlmClass.EOFF) OR (THIS^.checkAlmClassAllMultiChild(E_AlmClass.EOFF)) THEN
	CIf.Job.eMe_ActivAlmClass := E_AlmClass.EOFF;
	me.Alarm.bolfp := TRUE;
ELSIF (pRFW_CIF^.Job.eMe_ActivAlmClass=E_AlmClass.OFF) OR (THIS^.checkAlmClassAllMultiChild(E_AlmClass.OFF)) THEN
	CIf.Job.eMe_ActivAlmClass := E_AlmClass.OFF;
	me.Alarm.bolfp := TRUE;
ELSIF (pRFW_CIF^.Job.eMe_ActivAlmClass=E_AlmClass.STOP) OR (THIS^.checkAlmClassAllMultiChild(E_AlmClass.STOP)) THEN
	CIf.Job.eMe_ActivAlmClass := E_AlmClass.STOP;
	me.Alarm.bolfp := TRUE;
ELSE
	IF (me.Alarm.bolfp) THEN
		CIf.Job.eMe_ActivAlmClass := E_AlmClass.NONE; // no reset necessary
		me.Alarm.bolfp := FALSE;
	END_IF
END_IF

//------------------------------------------------------------------------------------------------------
// set alarm class parent of childs
IF (CIf.Job.eParent_ActivAlmClass=E_AlmClass.EOFF) OR (CIf.Job.eParent_ActivAlmClass=E_AlmClass.OFF) THEN
	pRFW_CIF^.Job.eParent_ActivAlmClass := CIf.Job.eParent_ActivAlmClass;
	THIS^.SetAlmClassAllMultiChild(CIf.Job.eParent_ActivAlmClass);
ELSIF(CIf.Job.eMe_ActivAlmClass=E_AlmClass.EOFF) OR (CIf.Job.eMe_ActivAlmClass=E_AlmClass.OFF) THEN
	pRFW_CIF^.Job.eParent_ActivAlmClass := CIf.Job.eMe_ActivAlmClass;
	THIS^.SetAlmClassAllMultiChild(CIf.Job.eMe_ActivAlmClass);
ELSE
	// no important alarm for child active
	pRFW_CIF^.Job.eParent_ActivAlmClass := E_AlmClass.NONE;
	THIS^.SetAlmClassAllMultiChild(E_AlmClass.NONE);
END_IF
END_METHOD

METHOD PROTECTED checkChildPointer : BOOL
IF (usiNumOfMultiChild = usiNumOfValidPointerMultiChild) THEN
	checkChildPointer:= TRUE;
ELSE
	checkChildPointer:= FALSE;
END_IF
END_METHOD

METHOD PROTECTED checkStateAllMultiChild : BOOL
VAR_INPUT
	cSTA: INT;
END_VAR
VAR
	ii: INT;
	usiNumOfCheckedChilds: USINT;
END_VAR
// Method check input state of all zones

//Init
checkStateAllMultiChild:= FALSE;
usiNumOfCheckedChilds:= 0;

// Loop over all childs
FOR ii:=0 TO usiNumOfMultiChild-1 BY 1 DO
	// Check state
	// Special condition: In case if the child is in state ERROR and STOP is requested. Set child as checked.
	// Parent controller need state STOP that automatic stop sequence can work for all other childs.
	IF (a_pMultiChildCIF[ii]^.Job.intState = cSTA) OR ((a_pMultiChildCIF[ii]^.Job.intState = cSTA_ERROR) AND (cSTA = cSTA_STOP)) THEN
		usiNumOfCheckedChilds:= usiNumOfCheckedChilds+1;
	END_IF

END_FOR

// All states equal the input state
IF (usiNumOfCheckedChilds = usiNumOfMultiChild) THEN
	checkStateAllMultiChild:= TRUE;
END_IF
END_METHOD

METHOD PROTECTED CmdToAllMultiChild
VAR_INPUT
	cCMD: INT;
END_VAR
VAR
	ii: INT;
END_VAR
// Method send input command to all existing multi child controller.
FOR ii:=0 TO usiNumOfMultiChild-1 BY 1 DO	
	a_pMultiChildCIF[ii]^.Job.intACmd:= cCMD;
END_FOR
END_METHOD

METHOD PROTECTED CtrlInit : BOOL
VAR
	ii: INT;
	usiChildIndex: USINT;
END_VAR
SUPER^.CtrlInit();

// get child common if
pRFW_CIf := p_fbRFW^.CtrlCIf;

// get specific interface for additional parmaeters or cur
pRFW_SIf := p_fbRFW^.getCtrlSIf();

//entry childs
usiChildIndex := 0;
THIS^.CIf.Info.p_aCIf[usiChildIndex] := THIS^.pRFW_CIf;
usiChildIndex := usiChildIndex+1;

// set parent id
pRFW_CIf^.Info.intParentCtrlId := CIf.Info.intCtrlId;

//initialize all multi Child controller.
FOR ii:=0 TO usiNumOfMultiChild-1 BY 1 DO	
	// Get child common if
	a_pMultiChildCIF[ii]:= a_pMultiChildCtrl[ii]^.CtrlCIf;	
	// Get specific interface for additional parmaeters or cur
	a_pMultiChildSIF[ii]:= a_pMultiChildCtrl[ii]^.getCtrlSIf();
	// Entry child
	THIS^.CIf.Info.p_aCIf[usiChildIndex]:= THIS^.a_pMultiChildCIF[ii];	
	usiChildIndex := usiChildIndex+1;
	// Set parent id
	a_pMultiChildCIF[ii]^.Info.intParentCtrlId := CIf.Info.intCtrlId;
	// Pointer to Hashtable
	a_pMultiChildSIF[ii]^.Par.pTblDecision := ADR(aTblDecision[0]);
	//*******************************************************************************
	// initial values childes
	//*******************************************************************************
	a_pMultiChildSIF[ii]^.Cfg.dinTargetNr := ii+1;
	//a_pMultiChildSIF[ii]^.Par.dinPosition_um := (ii+1) * 1000000;
END_FOR

// Determine the distance to the farthest (last) junction
SIf.Cur.dinDistanceToFarthestJunction:= 0;
FOR ii:=0 TO usiNumOfMultiChild-1 BY 1 DO
	IF (a_pMultiChildSIF[ii]^.Par.dinPosition_um > SIf.Cur.dinDistanceToFarthestJunction) THEN
		SIf.Cur.dinDistanceToFarthestJunction:= a_pMultiChildSIF[ii]^.Par.dinPosition_um;
	END_IF
END_FOR

SIf.Cfg.bolDtChToLine_send := TRUE;
END_METHOD

METHOD DtChnToPLC_Decision : BOOL
VAR
	bolRFIDExist: BOOL;
END_VAR
VAR CONSTANT
	cSTA_SUB_Data_Init: INT := 900;
	cSTA_SUB_Data_WaitForJob: INT := 902;
	cSTA_SUB_Data_CheckData: INT := 904;
	cSTA_SUB_Data_Acknowledge: INT := 906;
	cSTA_SUB_Data_Retry: INT := 908;
	cSTA_SUB_Data_Error: INT := 910;
	cDataState_Ready: INT := 1;
	cDataState_DONE: INT := -1;
	cDataState_Retry: INT := -99;
	cDataState_Error: INT := -100;
	cMAX_RETRY: INT := 10;
END_VAR
// Data Channel to Receive Data from Line Controller
// Startup check States
IF intStatemachine < cSTA_SUB_Data_Init THEN
	intStatemachine := cSTA_SUB_Data_Init;
END_IF

CASE intStatemachine OF
	cSTA_SUB_Data_Init:
		IF CIf.Job.intState > cSTA_PON THEN
			intCountRetry := 0;
			SIf.DtChnToPLC.stNewDecision.intDataState := cDataState_DONE;
			intStatemachine := cSTA_SUB_Data_WaitForJob;
		END_IF
		
	cSTA_SUB_Data_WaitForJob:
		// New data arrived
		IF SIf.DtChnToPLC.stNewDecision.intDataState = cDataState_Ready THEN
			bolDataBad := FALSE;
			dtOldestTag := dtActualTime;
			intIndexOldest := -1;			// -1 = no Oldest free input found
			intStatemachine := cSTA_SUB_Data_CheckData;
		END_IF
	
	cSTA_SUB_Data_CheckData:	
		// Check Data
		IF SIf.DtChnToPLC.stNewDecision.stDecision.uliRFID <= 0 THEN
				bolDataBad := TRUE;
				// Set Alarm: SIf.Alm[3].strText := 'False Job Parameter';
				pfbAlarmCtrl^.setAlarm(CIf.Info.intCtrlId,3,0,ADR(SIf.Alm),E_AlmState.RST,CIf.Job.eMe_ActivAlmClass);					
		END_IF 
		IF ((SIf.DtChnToPLC.stNewDecision.stDecision.dinTarget <= 0) OR
			 (SIf.DtChnToPLC.stNewDecision.stDecision.dinTarget > SIf.Cfg.intCountJunctions)) THEN
				bolDataBad := TRUE;
				// Set Alarm: SIf.Alm[3].strText := 'False Job Parameter';
				pfbAlarmCtrl^.setAlarm(CIf.Info.intCtrlId,3,SIf.DtChnToPLC.stNewDecision.stDecision.dinTarget,ADR(SIf.Alm),E_AlmState.RST,CIf.Job.eMe_ActivAlmClass);					
		END_IF 
		IF SIf.DtChnToPLC.stNewDecision.intJob <= E_Decision_Job.none AND SIf.DtChnToPLC.stNewDecision.intJob >= E_Decision_Job.MAX_E_Decision_Job THEN
				bolDataBad := TRUE;
				// Set Alarm: SIf.Alm[3].strText := 'False Job Parameter';
				pfbAlarmCtrl^.setAlarm(CIf.Info.intCtrlId,3,0,ADR(SIf.Alm),E_AlmState.RST,CIf.Job.eMe_ActivAlmClass);					
		END_IF 
		
				
		CASE SIf.DtChnToPLC.stNewDecision.intJob OF
			/////////////////////////////////////////////////////
			// Insert new decision item
			/////////////////////////////////////////////////////							
			E_Decision_Job.NEW:
				
				bolRFIDExist:= FALSE;
				//---------------------------------------
				// Loop through the hashtable
				//---------------------------------------
				FOR uinLoopRFID := 0 TO INT_TO_UINT(cintMaxDecisions) DO
					
					// Check if RFID already exist
					IF ((aTblDecision[uinLoopRFID].stDecision.uliRFID = SIf.DtChnToPLC.stNewDecision.stDecision.uliRFID) AND (bolRFIDExist=FALSE)) THEN
						// Save actual index of found RFID
						intIndexActualRFID := UINT_TO_INT(uinLoopRFID);				
						bolRFIDExist:= TRUE;
					END_IF	

					// In the same loop, save the index of the oldest input
					IF ((dtOldestTag > aTblDecision[uinLoopRFID].dtTimeJob) AND (aTblDecision[uinLoopRFID].eState = E_DecisionState.Finished)) THEN
						dtOldestTag := aTblDecision[uinLoopRFID].dtTimeJob;
						intIndexOldest := UINT_TO_INT(uinLoopRFID);
					END_IF
					
				END_FOR
				
				//---------------------------------------
				// Check bad data, retry handling
				//---------------------------------------
				IF bolDataBad = TRUE THEN
					IF intCountRetry >= cMAX_RETRY THEN
						intStatemachine := cSTA_SUB_Data_Error;
					ELSE
						intCountRetry := intCountRetry + 1;
						intStatemachine := cSTA_SUB_Data_Retry;
					END_IF
					
				//---------------------------------------
				// RFID already exist
				//---------------------------------------
				ELSIF bolRFIDExist THEN
					
					// In this case, the hanger is already on the way to junction.
					// Only now, the target is determined from line control!	
					aTblDecision[intIndexActualRFID].stDecision.dinTarget := SIf.DtChnToPLC.stNewDecision.stDecision.dinTarget;
					aTblDecision[intIndexActualRFID].dtTimeJob := dtActualTime;
					aTblDecision[intIndexActualRFID].eState := E_DecisionState.WayToJunction; // ????
					intStatemachine := cSTA_SUB_Data_Acknowledge;

			
				//---------------------------------------
				// RFID not exist
				//---------------------------------------
				ELSIF NOT(bolRFIDExist) THEN
					// Reset counter because right job
					intCountRetry := 0;
					
					// Search a free Element
					uinLoopRFID := 0;
					WHILE uinLoopRFID <= INT_TO_UINT(cintMaxDecisions) DO
						// NO RFID = Free element
						IF (aTblDecision[uinLoopRFID].stDecision.uliRFID = 0) THEN
							aTblDecision[uinLoopRFID].stDecision.uliRFID := SIf.DtChnToPLC.stNewDecision.stDecision.uliRFID;
							aTblDecision[uinLoopRFID].stDecision.dinTarget := SIf.DtChnToPLC.stNewDecision.stDecision.dinTarget;
							aTblDecision[uinLoopRFID].dtTimeJob := dtActualTime;
							aTblDecision[uinLoopRFID].eState := E_DecisionState.Wait;						
							intStatemachine := cSTA_SUB_Data_Acknowledge;
							EXIT;
						END_IF
					
						uinLoopRFID := uinLoopRFID + 1;	
					END_WHILE
					
					// IF Loop was finished and no input done = No empty Hashtable line was there
					// Overwrite the oldest one                   
					IF ((UINT_TO_INT(uinLoopRFID) = cintMaxDecisions) AND (aTblDecision[uinLoopRFID].stDecision.uliRFID <> SIf.DtChnToPLC.stNewDecision.stDecision.uliRFID)) THEN
						// The oldest input was saved at a loop before
						IF intIndexOldest >= 0 THEN		// A possible line to overwrite was found: -1 = initial value
							aTblDecision[intIndexOldest].stDecision.uliRFID := SIf.DtChnToPLC.stNewDecision.stDecision.uliRFID;
							aTblDecision[intIndexOldest].stDecision.dinTarget := SIf.DtChnToPLC.stNewDecision.stDecision.dinTarget;
							aTblDecision[intIndexOldest].dtTimeJob := dtActualTime;
							aTblDecision[intIndexOldest].eState := E_DecisionState.Wait;
							intStatemachine := cSTA_SUB_Data_Acknowledge;
						ELSE
							intStatemachine := cDataState_Error;		// No other inputs are possible
							// Set Alarm: SIf.Alm[7].strText := 'Hashtable full, no more input possible';
							pfbAlarmCtrl^.setAlarm(CIf.Info.intCtrlId,7,cintMaxDecisions,ADR(SIf.Alm),E_AlmState.RST,CIf.Job.eMe_ActivAlmClass);										
						END_IF
					END_IF
				END_IF
				
			/////////////////////////////////////////////////////
			// Replace ID
			/////////////////////////////////////////////////////			
			E_Decision_Job.REPLACE_ID:
				// Init value
				bolDataFound := FALSE;
				// Check if RF ID not allready exist
				FOR uinLoopRFID := 0 TO INT_TO_UINT(cintMaxDecisions) DO
					IF aTblDecision[uinLoopRFID].stDecision.uliRFID = SIf.DtChnToPLC.stNewDecision.stDecision.uliRFID THEN
						aTblDecision[uinLoopRFID].stDecision.dinTarget := SIf.DtChnToPLC.stNewDecision.stDecision.dinTarget;
						aTblDecision[uinLoopRFID].dtTimeJob := dtActualTime;	
						bolDataFound := TRUE;					
						intStatemachine := cSTA_SUB_Data_Acknowledge;
						EXIT;
					END_IF
				END_FOR
				
				IF bolDataFound = FALSE THEN
					//Set Alarm: SIf.Alm[10].strText := 'RFID Not found';
					pfbAlarmCtrl^.setAlarm(CIf.Info.intCtrlId,10,0,ADR(SIf.Alm),E_AlmState.RST,CIf.Job.eMe_ActivAlmClass);					
					IF intCountRetry >= cMAX_RETRY THEN
						intStatemachine := cSTA_SUB_Data_Error;
					ELSE
						intCountRetry := intCountRetry + 1;
						intStatemachine := cSTA_SUB_Data_Retry;
					END_IF
				END_IF

			/////////////////////////////////////////////////////
			// Delete ID
			/////////////////////////////////////////////////////			
			E_Decision_Job.DELETE_ID:
				// Init value
				bolDataFound := FALSE;
				// Check if RF ID not allready exist
				FOR uinLoopRFID := 0 TO INT_TO_UINT(cintMaxDecisions) DO
					IF aTblDecision[uinLoopRFID].stDecision.uliRFID = SIf.DtChnToPLC.stNewDecision.stDecision.uliRFID THEN
						// Check DecisionState before delete
						IF (aTblDecision[uinLoopRFID].eState = E_DecisionState.Wait) OR 
							(aTblDecision[uinLoopRFID].eState = E_DecisionState.WayToJunction) OR
							(aTblDecision[uinLoopRFID].eState = E_DecisionState.Finished) THEN
 
							aTblDecision[uinLoopRFID].stDecision.uliRFID := 0;
							aTblDecision[uinLoopRFID].stDecision.dinTarget := 0;
							aTblDecision[uinLoopRFID].dtTimeJob := DINT_TO_DT(0);
							aTblDecision[uinLoopRFID].eState := E_DecisionState.none;
							aTblDecision[uinLoopRFID].dinActPos_um := 0;
							aTblDecision[uinLoopRFID].dtTimeRFID := DINT_TO_DT(0);
						
							intStatemachine := cSTA_SUB_Data_Acknowledge;
							bolDataFound := TRUE;					
							EXIT;
						END_IF
					END_IF
				END_FOR
				
				IF bolDataFound = FALSE THEN
					//Set Alarm: SIf.Alm[10].strText := 'RFID Not found';
					pfbAlarmCtrl^.setAlarm(CIf.Info.intCtrlId,10,0,ADR(SIf.Alm),E_AlmState.RST,CIf.Job.eMe_ActivAlmClass);					
					IF intCountRetry >= cMAX_RETRY THEN
						intStatemachine := cSTA_SUB_Data_Error;
					ELSE
						intCountRetry := intCountRetry + 1;
						intStatemachine := cSTA_SUB_Data_Retry;
					END_IF
				END_IF
				
			/////////////////////////////////////////////////////
			// Delete Junction
			/////////////////////////////////////////////////////			
			E_Decision_Job.DELETE_JUNCTION:
				// Check if RF ID not allready exist
				FOR uinLoopRFID := 0 TO INT_TO_UINT(cintMaxDecisions) DO
					IF aTblDecision[uinLoopRFID].stDecision.dinTarget = SIf.DtChnToPLC.stNewDecision.stDecision.dinTarget THEN
						// Check DecisionState before delete junction
						IF (aTblDecision[uinLoopRFID].eState = E_DecisionState.Wait) OR 
							(aTblDecision[uinLoopRFID].eState = E_DecisionState.WayToJunction) OR
							(aTblDecision[uinLoopRFID].eState = E_DecisionState.Finished) THEN
							
